LIN {X 0,Y 366.186,Z 582.317,A -85,B 0,C 180,E1 11317.948,E2 11317.948} C_VEL
LIN {X 0,Y 371.431,Z 589.202,A -85,B 0,C 180,E1 11315.424,E2 11315.424} C_VEL
LIN {X 0,Y 378.008,Z 597.97,A -85,B 0,C 180,E1 11312.682,E2 11312.682} C_VEL
LIN {X 0,Y 385.262,Z 608.266,A -85,B 0,C 180,E1 11310.027,E2 11310.027} C_VEL
LIN {X 0,Y 392.759,Z 619.158,A -85,B 0,C 180,E1 11307.596,E2 11307.596} C_VEL
LIN {X 0,Y 401.924,Z 633.691,A -85,B 0,C 180,E1 11304.924,E2 11304.924} C_VEL
LIN {X 0,Y 408.714,Z 645.3,A -85,B 0,C 180,E1 11303.115,E2 11303.115} C_VEL
LIN {X 0,Y 397.678,Z 876.786,A -85,B 0,C 180,E1 11298.792,E2 11298.792} C_VEL
LIN {X 0,Y 395.952,Z 903.504,A -85,B 0,C 180,E1 11298.228,E2 11298.228} C_VEL
LIN {X 0,Y 393.493,Z 925.311,A -85,B 0,C 180,E1 11297.568,E2 11297.568} C_VEL
LIN {X 0,Y 390.28,Z 946.189,A -85,B 0,C 180,E1 11296.684,E2 11296.684} C_VEL
LIN {X 0,Y 386.282,Z 967.256,A -85,B 0,C 180,E1 11295.529,E2 11295.529} C_VEL
LIN {X 0,Y 382.072,Z 986.142,A -85,B 0,C 180,E1 11294.243,E2 11294.243} C_VEL
LIN {X 0,Y 377.137,Z 1005.209,A -85,B 0,C 180,E1 11292.639,E2 11292.639} C_VEL
LIN {X 0,Y 371.736,Z 1024.131,A -85,B 0,C 180,E1 11290.712,E2 11290.712} C_VEL
LIN {X 0,Y 366.371,Z 1041.49,A -85,B 0,C 180,E1 11288.579,E2 11288.579} C_VEL
LIN {X 0,Y 361.104,Z 1057.311,A -85,B 0,C 180,E1 11286.24,E2 11286.24} C_VEL
LIN {X 0,Y 355.944,Z 1072.38,A -85,B 0,C 180,E1 11283.599,E2 11283.599} C_VEL
LIN {X 0,Y 351.082,Z 1086.425,A -85,B 0,C 180,E1 11280.649,E2 11280.649} C_VEL
LIN {X 0,Y 346.966,Z 1098.332,A -85,B 0,C 180,E1 11277.643,E2 11277.643} C_VEL
LIN {X 0,Y 343.299,Z 1109.594,A -85,B 0,C 180,E1 11274.247,E2 11274.247} C_VEL
LIN {X 0,Y 340.505,Z 1118.917,A -85,B 0,C 180,E1 11270.812,E2 11270.812} C_VEL
LIN {X 0,Y 338.432,Z 1126.851,A -85,B 0,C 180,E1 11267.184,E2 11267.184} C_VEL
LIN {X 0,Y 337.113,Z 1133.168,A -85,B 0,C 180,E1 11263.551,E2 11263.551} C_VEL
LIN {X 0,Y 336.408,Z 1137.619,A -85,B 0,C 180,E1 11260.099,E2 11260.099} C_VEL
LIN {X 0,Y 336.159,Z 1139.83,A -85,B 0,C 180,E1 11257.841,E2 11257.841} C_VEL
LIN {X 0,Y 335.071,Z 1140.944,A -85,B 0,C 180,E1 11256.542,E2 11256.542} C_VEL
LIN {X 0,Y 330.367,Z 1142.612,A -85,B 0,C 180,E1 11254.081,E2 11254.081} C_VEL
LIN {X 0,Y 328.115,Z 1143.242,A -85,B 0,C 180,E1 11252.372,E2 11252.372} C_VEL
LIN {X 0,Y 327.966,Z 1143.315,A -85,B 0,C 180,E1 11251.884,E2 11251.884} C_VEL
LIN {X 0,Y 327.969,Z 1143.385,A -85,B 0,C 180,E1 11248.602,E2 11248.602} C_VEL
LIN {X 0,Y 328.018,Z 1142.229,A -85,B 0,C 180,E1 11244.929,E2 11244.929} C_VEL
LIN {X 0,Y 328.248,Z 1139.737,A -85,B 0,C 180,E1 11241.416,E2 11241.416} C_VEL
LIN {X 0,Y 328.872,Z 1135.354,A -85,B 0,C 180,E1 11237.404,E2 11237.404} C_VEL
LIN {X 0,Y 330.06,Z 1129.659,A -85,B 0,C 180,E1 11233.637,E2 11233.637} C_VEL
LIN {X 0,Y 331.98,Z 1122.268,A -85,B 0,C 180,E1 11229.919,E2 11229.919} C_VEL
LIN {X 0,Y 334.944,Z 1112.65,A -85,B 0,C 180,E1 11226.047,E2 11226.047} C_VEL
LIN {X 0,Y 338.59,Z 1102.053,A -85,B 0,C 180,E1 11222.57,E2 11222.57} C_VEL
LIN {X 0,Y 342.919,Z 1089.92,A -85,B 0,C 180,E1 11219.319,E2 11219.319} C_VEL
LIN {X 0,Y 347.843,Z 1076.454,A -85,B 0,C 180,E1 11216.305,E2 11216.305} C_VEL
LIN {X 0,Y 353.24,Z 1061.666,A -85,B 0,C 180,E1 11213.529,E2 11213.529} C_VEL
LIN {X 0,Y 358.581,Z 1046.318,A -85,B 0,C 180,E1 11211.142,E2 11211.142} C_VEL
LIN {X 0,Y 364.459,Z 1028.526,A -85,B 0,C 180,E1 11208.82,E2 11208.82} C_VEL
LIN {X 0,Y 370.03,Z 1010.354,A -85,B 0,C 180,E1 11206.851,E2 11206.851} C_VEL
LIN {X 0,Y 375.194,Z 991.424,A -85,B 0,C 180,E1 11205.181,E2 11205.181} C_VEL
LIN {X 0,Y 380.213,Z 970.596,A -85,B 0,C 180,E1 11203.682,E2 11203.682} C_VEL
LIN {X 0,Y 384.198,Z 951.289,A -85,B 0,C 180,E1 11202.566,E2 11202.566} C_VEL
LIN {X 0,Y 387.659,Z 930.348,A -85,B 0,C 180,E1 11201.626,E2 11201.626} C_VEL
LIN {X 0,Y 390.429,Z 909.023,A -85,B 0,C 180,E1 11200.912,E2 11200.912} C_VEL
LIN {X 0,Y 392.234,Z 887.054,A -85,B 0,C 180,E1 11200.398,E2 11200.398} C_VEL
LIN {X 0,Y 400.836,Z 709.616,A -85,B 0,C 180,E1 11197.043,E2 11197.043} C_VEL
LIN {X 0,Y 396.954,Z 714.225,A -85,B 0,C 180,E1 11196.361,E2 11196.361} C_VEL
LIN {X 0,Y 391.32,Z 723.362,A -85,B 0,C 180,E1 11195.402,E2 11195.402} C_VEL
LIN {X 0,Y 386.047,Z 730.128,A -85,B 0,C 180,E1 11194.399,E2 11194.399} C_VEL
LIN {X 0,Y 380.733,Z 739.752,A -85,B 0,C 180,E1 11193.425,E2 11193.425} C_VEL
LIN {X 0,Y 377.937,Z 744.145,A -85,B 0,C 180,E1 11192.866,E2 11192.866} C_VEL
LIN {X 0,Y 373.251,Z 764.172,A -85,B 0,C 180,E1 11192.35,E2 11192.35} C_VEL
LIN {X 0,Y 369.775,Z 775.752,A -85,B 0,C 180,E1 11191.833,E2 11191.833} C_VEL
LIN {X 0,Y 367.625,Z 781.787,A -85,B 0,C 180,E1 11191.463,E2 11191.463} C_VEL
LIN {X 0,Y 361.181,Z 811.219,A -85,B 0,C 180,E1 11190.749,E2 11190.749} C_VEL
LIN {X 0,Y 357.761,Z 823.668,A -85,B 0,C 180,E1 11190.226,E2 11190.226} C_VEL
LIN {X 0,Y 354.98,Z 831.573,A -85,B 0,C 180,E1 11189.695,E2 11189.695} C_VEL
LIN {X 0,Y 348.335,Z 862.323,A -85,B 0,C 180,E1 11188.874,E2 11188.874} C_VEL
LIN {X 0,Y 345.171,Z 873.899,A -85,B 0,C 180,E1 11188.328,E2 11188.328} C_VEL
LIN {X 0,Y 343.261,Z 880.377,A -85,B 0,C 180,E1 11187.812,E2 11187.812} C_VEL
LIN {X 0,Y 342.63,Z 889.884,A -85,B 0,C 180,E1 11187.433,E2 11187.433} C_VEL
LIN {X 0,Y 342.059,Z 911.963,A -85,B 0,C 180,E1 11186.73,E2 11186.73} C_VEL
LIN {X 0,Y 341.208,Z 929.996,A -85,B 0,C 180,E1 11185.842,E2 11185.842} C_VEL
LIN {X 0,Y 339.993,Z 948.311,A -85,B 0,C 180,E1 11184.591,E2 11184.591} C_VEL
LIN {X 0,Y 338.687,Z 963.946,A -85,B 0,C 180,E1 11183.211,E2 11183.211} C_VEL
LIN {X 0,Y 337.194,Z 979.445,A -85,B 0,C 180,E1 11181.482,E2 11181.482} C_VEL
LIN {X 0,Y 335.66,Z 993.949,A -85,B 0,C 180,E1 11179.489,E2 11179.489} C_VEL
LIN {X 0,Y 334.281,Z 1006.231,A -85,B 0,C 180,E1 11177.404,E2 11177.404} C_VEL
LIN {X 0,Y 332.98,Z 1017.915,A -85,B 0,C 180,E1 11174.966,E2 11174.966} C_VEL
LIN {X 0,Y 332,Z 1027.395,A -85,B 0,C 180,E1 11172.524,E2 11172.524} C_VEL
LIN {X 0,Y 331.241,Z 1035.395,A -85,B 0,C 180,E1 11169.908,E2 11169.908} C_VEL
LIN {X 0,Y 330.761,Z 1041.946,A -85,B 0,C 180,E1 11167.12,E2 11167.12} C_VEL
LIN {X 0,Y 330.565,Z 1046.667,A -85,B 0,C 180,E1 11164.337,E2 11164.337} C_VEL
LIN {X 0,Y 330.581,Z 1049.61,A -85,B 0,C 180,E1 11161.56,E2 11161.56} C_VEL
LIN {X 0,Y 330.804,Z 1050.944,A -85,B 0,C 180,E1 11158.615,E2 11158.615} C_VEL
LIN {X 0,Y 331.202,Z 1050.526,A -85,B 0,C 180,E1 11155.846,E2 11155.846} C_VEL
LIN {X 0,Y 331.838,Z 1048.398,A -85,B 0,C 180,E1 11153.078,E2 11153.078} C_VEL
LIN {X 0,Y 332.756,Z 1044.468,A -85,B 0,C 180,E1 11150.313,E2 11150.313} C_VEL
LIN {X 0,Y 334.013,Z 1038.61,A -85,B 0,C 180,E1 11147.554,E2 11147.554} C_VEL
LIN {X 0,Y 335.392,Z 1031.672,A -85,B 0,C 180,E1 11145.145,E2 11145.145} C_VEL
LIN {X 0,Y 337.024,Z 1022.654,A -85,B 0,C 180,E1 11142.743,E2 11142.743} C_VEL
LIN {X 0,Y 338.799,Z 1012.138,A -85,B 0,C 180,E1 11140.52,E2 11140.52} C_VEL
LIN {X 0,Y 340.605,Z 999.902,A -85,B 0,C 180,E1 11138.473,E2 11138.473} C_VEL
LIN {X 0,Y 342.308,Z 986.562,A -85,B 0,C 180,E1 11136.686,E2 11136.686} C_VEL
LIN {X 0,Y 343.887,Z 971.383,A -85,B 0,C 180,E1 11135.066,E2 11135.066} C_VEL
LIN {X 0,Y 345.235,Z 954.859,A -85,B 0,C 180,E1 11133.698,E2 11133.698} C_VEL
LIN {X 0,Y 346.219,Z 937.734,A -85,B 0,C 180,E1 11132.62,E2 11132.62} C_VEL
LIN {X 0,Y 346.855,Z 927.468,A -85,B 0,C 180,E1 11132.068,E2 11132.068} C_VEL
LIN {X 0,Y 348,Z 924.934,A -85,B 0,C 180,E1 11131.772,E2 11131.772} C_VEL
LIN {X 0,Y 350.86,Z 920.539,A -85,B 0,C 180,E1 11131.345,E2 11131.345} C_VEL
LIN {X 0,Y 354.501,Z 912.006,A -85,B 0,C 180,E1 11131.007,E2 11131.007} C_VEL
LIN {X 0,Y 357.108,Z 904.907,A -85,B 0,C 180,E1 11130.799,E2 11130.799} C_VEL
LIN {X 0,Y 360.337,Z 898.788,A -85,B 0,C 180,E1 11130.331,E2 11130.331} C_VEL
LIN {X 0,Y 363.987,Z 888.542,A -85,B 0,C 180,E1 11129.925,E2 11129.925} C_VEL
LIN {X 0,Y 369.949,Z 866.042,A -85,B 0,C 180,E1 11129.35,E2 11129.35} C_VEL
LIN {X 0,Y 373.838,Z 855.883,A -85,B 0,C 180,E1 11128.8,E2 11128.8} C_VEL
LIN {X 0,Y 378.866,Z 838.681,A -85,B 0,C 180,E1 11128.259,E2 11128.259} C_VEL
LIN {X 0,Y 383.059,Z 822.695,A -85,B 0,C 180,E1 11127.883,E2 11127.883} C_VEL
LIN {X 0,Y 387.383,Z 811.4,A -85,B 0,C 180,E1 11127.333,E2 11127.333} C_VEL
LIN {X 0,Y 392.621,Z 793.713,A -85,B 0,C 180,E1 11126.825,E2 11126.825} C_VEL
LIN {X 0,Y 396.512,Z 779.247,A -85,B 0,C 180,E1 11126.502,E2 11126.502} C_VEL
LIN {X 0,Y 399.615,Z 771.69,A -85,B 0,C 180,E1 11126.126,E2 11126.126} C_VEL
LIN {X 0,Y 392.671,Z 892.302,A -85,B 0,C 180,E1 11123.671,E2 11123.671} C_VEL
LIN {X 0,Y 390.102,Z 915.62,A -85,B 0,C 180,E1 11123.008,E2 11123.008} C_VEL
LIN {X 0,Y 386.994,Z 937.185,A -85,B 0,C 180,E1 11122.181,E2 11122.181} C_VEL
LIN {X 0,Y 382.98,Z 959.044,A -85,B 0,C 180,E1 11121.078,E2 11121.078} C_VEL
LIN {X 0,Y 378.27,Z 980.989,A -85,B 0,C 180,E1 11119.696,E2 11119.696} C_VEL
LIN {X 0,Y 373.314,Z 1001.28,A -85,B 0,C 180,E1 11118.123,E2 11118.123} C_VEL
LIN {X 0,Y 367.979,Z 1020.909,A -85,B 0,C 180,E1 11116.284,E2 11116.284} C_VEL
LIN {X 0,Y 362.493,Z 1039.821,A -85,B 0,C 180,E1 11114.181,E2 11114.181} C_VEL
LIN {X 0,Y 356.917,Z 1057.605,A -85,B 0,C 180,E1 11111.815,E2 11111.815} C_VEL
LIN {X 0,Y 351.301,Z 1075.094,A -85,B 0,C 180,E1 11109.082,E2 11109.082} C_VEL
LIN {X 0,Y 346.378,Z 1090.22,A -85,B 0,C 180,E1 11106.282,E2 11106.282} C_VEL
LIN {X 0,Y 341.513,Z 1105.32,A -85,B 0,C 180,E1 11102.995,E2 11102.995} C_VEL
LIN {X 0,Y 337.534,Z 1118.368,A -85,B 0,C 180,E1 11099.65,E2 11099.65} C_VEL
LIN {X 0,Y 334.214,Z 1129.964,A -85,B 0,C 180,E1 11096.09,E2 11096.09} C_VEL
LIN {X 0,Y 331.63,Z 1140.317,A -85,B 0,C 180,E1 11092.327,E2 11092.327} C_VEL
LIN {X 0,Y 329.914,Z 1148.379,A -85,B 0,C 180,E1 11088.739,E2 11088.739} C_VEL
LIN {X 0,Y 328.748,Z 1155.565,A -85,B 0,C 180,E1 11084.802,E2 11084.802} C_VEL
LIN {X 0,Y 328.211,Z 1160.559,A -85,B 0,C 180,E1 11081.209,E2 11081.209} C_VEL
LIN {X 0,Y 327.959,Z 1164.449,A -85,B 0,C 180,E1 11077.357,E2 11077.357} C_VEL
LIN {X 0,Y 327.941,Z 1166.518,A -85,B 0,C 180,E1 11073.846,E2 11073.846} C_VEL
LIN {X 0,Y 327.936,Z 1167.332,A -85,B 0,C 180,E1 11070.524,E2 11070.524} C_VEL
LIN {X 0,Y 327.927,Z 1166.805,A -85,B 0,C 180,E1 11066.854,E2 11066.854} C_VEL
LIN {X 0,Y 327.965,Z 1165.053,A -85,B 0,C 180,E1 11063.523,E2 11063.523} C_VEL
LIN {X 0,Y 328.1,Z 1161.814,A -85,B 0,C 180,E1 11059.819,E2 11059.819} C_VEL
LIN {X 0,Y 328.575,Z 1156.905,A -85,B 0,C 180,E1 11056.09,E2 11056.09} C_VEL
LIN {X 0,Y 329.54,Z 1150.522,A -85,B 0,C 180,E1 11052.307,E2 11052.307} C_VEL
LIN {X 0,Y 331.12,Z 1142.434,A -85,B 0,C 180,E1 11048.569,E2 11048.569} C_VEL
LIN {X 0,Y 333.509,Z 1132.644,A -85,B 0,C 180,E1 11044.804,E2 11044.804} C_VEL
LIN {X 0,Y 336.436,Z 1121.99,A -85,B 0,C 180,E1 11041.414,E2 11041.414} C_VEL
LIN {X 0,Y 340.395,Z 1108.935,A -85,B 0,C 180,E1 11037.882,E2 11037.882} C_VEL
LIN {X 0,Y 344.735,Z 1095.225,A -85,B 0,C 180,E1 11034.748,E2 11034.748} C_VEL
LIN {X 0,Y 349.892,Z 1079.355,A -85,B 0,C 180,E1 11031.676,E2 11031.676} C_VEL
LIN {X 0,Y 355.227,Z 1062.965,A -85,B 0,C 180,E1 11028.967,E2 11028.967} C_VEL
LIN {X 0,Y 360.826,Z 1044.991,A -85,B 0,C 180,E1 11026.48,E2 11026.48} C_VEL
LIN {X 0,Y 366.707,Z 1025.329,A -85,B 0,C 180,E1 11024.185,E2 11024.185} C_VEL
LIN {X 0,Y 371.762,Z 1007.076,A -85,B 0,C 180,E1 11022.396,E2 11022.396} C_VEL
LIN {X 0,Y 377.049,Z 986.011,A -85,B 0,C 180,E1 11020.675,E2 11020.675} C_VEL
LIN {X 0,Y 381.795,Z 964.869,A -85,B 0,C 180,E1 11019.258,E2 11019.258} C_VEL
LIN {X 0,Y 385.904,Z 942.947,A -85,B 0,C 180,E1 11018.093,E2 11018.093} C_VEL
LIN {X 0,Y 389.526,Z 919.577,A -85,B 0,C 180,E1 11017.128,E2 11017.128} C_VEL
LIN {X 0,Y 392.156,Z 897.248,A -85,B 0,C 180,E1 11016.458,E2 11016.458} C_VEL
LIN {X 0,Y 394.386,Z 863.932,A -85,B 0,C 180,E1 11015.736,E2 11015.736} C_VEL
LIN {X 0,Y 406.266,Z 655.335,A -85,B 0,C 180,E1 11011.555,E2 11011.555} C_VEL
LIN {X 0,Y 406.902,Z 643.594,A -85,B 0,C 180,E1 11011.312,E2 11011.312} C_VEL
LIN {X 0,Y 397.581,Z 629.012,A -85,B 0,C 180,E1 11008.748,E2 11008.748} C_VEL
LIN {X 0,Y 388.35,Z 615.637,A -85,B 0,C 180,E1 11005.915,E2 11005.915} C_VEL
LIN {X 0,Y 380.432,Z 605.01,A -85,B 0,C 180,E1 11003.177,E2 11003.177} C_VEL
LIN {X 0,Y 373.333,Z 595.852,A -85,B 0,C 180,E1 11000.375,E2 11000.375} C_VEL
LIN {X 0,Y 368.267,Z 589.841,A -85,B 0,C 180,E1 10998.111,E2 10998.111} C_VEL
LIN {X 0,Y 363.853,Z 584.59,A -85,B 0,C 180,E1 10995.868,E2 10995.868} C_VEL
LIN {X 0,Y 358.835,Z 578.864,A -85,B 0,C 180,E1 10992.88,E2 10992.88} C_VEL
LIN {X 0,Y 353.311,Z 572.841,A -85,B 0,C 180,E1 10988.626,E2 10988.626} C_VEL
LIN {X 0,Y 348.081,Z 567.999,A -85,B 0,C 180,E1 10981.646,E2 10981.646} C_VEL
LIN {X 0,Y 347.245,Z 567.182,A -85,B 0,C 180,E1 10978.184,E2 10978.184} C_VEL
LIN {X 0,Y 347.496,Z 568.254,A -85,B 0,C 180,E1 10974.551,E2 10974.551} C_VEL
LIN {X 0,Y 351.064,Z 572.556,A -85,B 0,C 180,E1 10968.166,E2 10968.166} C_VEL
LIN {X 0,Y 354.487,Z 577.164,A -85,B 0,C 180,E1 10964.792,E2 10964.792} C_VEL
LIN {X 0,Y 355.794,Z 578.575,A -85,B 0,C 180,E1 10963.762,E2 10963.762} C_VEL
LIN {X 0,Y 359.364,Z 583.21,A -85,B 0,C 180,E1 10961.255,E2 10961.255} C_VEL
LIN {X 0,Y 364.436,Z 589.819,A -85,B 0,C 180,E1 10958.303,E2 10958.303} C_VEL
LIN {X 0,Y 369.585,Z 596.701,A -85,B 0,C 180,E1 10955.761,E2 10955.761} C_VEL
LIN {X 0,Y 376.05,Z 605.555,A -85,B 0,C 180,E1 10952.999,E2 10952.999} C_VEL
LIN {X 0,Y 382.814,Z 615.312,A -85,B 0,C 180,E1 10950.462,E2 10950.462} C_VEL
LIN {X 0,Y 389.968,Z 625.925,A -85,B 0,C 180,E1 10948.076,E2 10948.076} C_VEL
LIN {X 0,Y 398.766,Z 640.106,A -85,B 0,C 180,E1 10945.438,E2 10945.438} C_VEL
LIN {X 0,Y 404.034,Z 649.281,A -85,B 0,C 180,E1 10943.979,E2 10943.979} C_VEL
LIN {X 0,Y 392.554,Z 879.807,A -85,B 0,C 180,E1 10939.647,E2 10939.647} C_VEL
LIN {X 0,Y 390.832,Z 904.21,A -85,B 0,C 180,E1 10939.118,E2 10939.118} C_VEL
LIN {X 0,Y 388.219,Z 926.195,A -85,B 0,C 180,E1 10938.44,E2 10938.44} C_VEL
LIN {X 0,Y 384.946,Z 946.674,A -85,B 0,C 180,E1 10937.567,E2 10937.567} C_VEL
LIN {X 0,Y 380.888,Z 967.279,A -85,B 0,C 180,E1 10936.429,E2 10936.429} C_VEL
LIN {X 0,Y 376.38,Z 986.786,A -85,B 0,C 180,E1 10935.094,E2 10935.094} C_VEL
LIN {X 0,Y 371.267,Z 1005.752,A -85,B 0,C 180,E1 10933.479,E2 10933.479} C_VEL
LIN {X 0,Y 365.653,Z 1024.604,A -85,B 0,C 180,E1 10931.537,E2 10931.537} C_VEL
LIN {X 0,Y 360.07,Z 1041.94,A -85,B 0,C 180,E1 10929.384,E2 10929.384} C_VEL
LIN {X 0,Y 354.594,Z 1057.668,A -85,B 0,C 180,E1 10927.024,E2 10927.024} C_VEL
LIN {X 0,Y 349.176,Z 1072.757,A -85,B 0,C 180,E1 10924.34,E2 10924.34} C_VEL
LIN {X 0,Y 344.328,Z 1086.047,A -85,B 0,C 180,E1 10921.513,E2 10921.513} C_VEL
LIN {X 0,Y 339.729,Z 1098.679,A -85,B 0,C 180,E1 10918.284,E2 10918.284} C_VEL
LIN {X 0,Y 335.848,Z 1109.925,A -85,B 0,C 180,E1 10914.82,E2 10914.82} C_VEL
LIN {X 0,Y 332.874,Z 1119.245,A -85,B 0,C 180,E1 10911.312,E2 10911.312} C_VEL
LIN {X 0,Y 330.651,Z 1127.166,A -85,B 0,C 180,E1 10907.601,E2 10907.601} C_VEL
LIN {X 0,Y 329.229,Z 1133.474,A -85,B 0,C 180,E1 10903.882,E2 10903.882} C_VEL
LIN {X 0,Y 328.457,Z 1137.92,A -85,B 0,C 180,E1 10900.347,E2 10900.347} C_VEL
LIN {X 0,Y 328.095,Z 1141.313,A -85,B 0,C 180,E1 10896.474,E2 10896.474} C_VEL
LIN {X 0,Y 327.975,Z 1143.026,A -85,B 0,C 180,E1 10892.971,E2 10892.971} C_VEL
LIN {X 0,Y 327.966,Z 1143.315,A -85,B 0,C 180,E1 10891.884,E2 10891.884} C_VEL
LIN {X 0,Y 326.958,Z 1143.526,A -85,B 0,C 180,E1 10890.538,E2 10890.538} C_VEL
LIN {X 0,Y 322.684,Z 1143.537,A -85,B 0,C 180,E1 10888.184,E2 10888.184} C_VEL
LIN {X 0,Y 320.264,Z 1143.171,A -85,B 0,C 180,E1 10886.435,E2 10886.435} C_VEL
LIN {X 0,Y 320.013,Z 1142.918,A -85,B 0,C 180,E1 10885.736,E2 10885.736} C_VEL
LIN {X 0,Y 320.204,Z 1140.562,A -85,B 0,C 180,E1 10881.834,E2 10881.834} C_VEL
LIN {X 0,Y 320.744,Z 1136.958,A -85,B 0,C 180,E1 10878.127,E2 10878.127} C_VEL
LIN {X 0,Y 321.813,Z 1131.693,A -85,B 0,C 180,E1 10874.317,E2 10874.317} C_VEL
LIN {X 0,Y 323.691,Z 1124.701,A -85,B 0,C 180,E1 10870.412,E2 10870.412} C_VEL
LIN {X 0,Y 326.349,Z 1116.278,A -85,B 0,C 180,E1 10866.72,E2 10866.72} C_VEL
LIN {X 0,Y 329.869,Z 1106.265,A -85,B 0,C 180,E1 10863.151,E2 10863.151} C_VEL
LIN {X 0,Y 334.125,Z 1095.008,A -85,B 0,C 180,E1 10859.819,E2 10859.819} C_VEL
LIN {X 0,Y 338.965,Z 1082.307,A -85,B 0,C 180,E1 10856.725,E2 10856.725} C_VEL
LIN {X 0,Y 344.643,Z 1067.47,A -85,B 0,C 180,E1 10853.713,E2 10853.713} C_VEL
LIN {X 0,Y 350.375,Z 1052.151,A -85,B 0,C 180,E1 10851.111,E2 10851.111} C_VEL
LIN {X 0,Y 356.201,Z 1035.575,A -85,B 0,C 180,E1 10848.789,E2 10848.789} C_VEL
LIN {X 0,Y 362.114,Z 1017.486,A -85,B 0,C 180,E1 10846.674,E2 10846.674} C_VEL
LIN {X 0,Y 367.65,Z 999.07,A -85,B 0,C 180,E1 10844.89,E2 10844.89} C_VEL
LIN {X 0,Y 372.724,Z 979.661,A -85,B 0,C 180,E1 10843.366,E2 10843.366} C_VEL
LIN {X 0,Y 377.633,Z 958.028,A -85,B 0,C 180,E1 10842.001,E2 10842.001} C_VEL
LIN {X 0,Y 381.486,Z 937.643,A -85,B 0,C 180,E1 10840.989,E2 10840.989} C_VEL
LIN {X 0,Y 384.509,Z 916.783,A -85,B 0,C 180,E1 10840.216,E2 10840.216} C_VEL
LIN {X 0,Y 386.877,Z 893.893,A -85,B 0,C 180,E1 10839.609,E2 10839.609} C_VEL
LIN {X 0,Y 395.423,Z 726.724,A -85,B 0,C 180,E1 10836.412,E2 10836.412} C_VEL
LIN {X 0,Y 389.741,Z 734.274,A -85,B 0,C 180,E1 10835.391,E2 10835.391} C_VEL
LIN {X 0,Y 388.254,Z 736.358,A -85,B 0,C 180,E1 10835.118,E2 10835.118} C_VEL
LIN {X 0,Y 382.655,Z 746.09,A -85,B 0,C 180,E1 10834.112,E2 10834.112} C_VEL
LIN {X 0,Y 381.204,Z 748.533,A -85,B 0,C 180,E1 10833.84,E2 10833.84} C_VEL
LIN {X 0,Y 376.48,Z 768.015,A -85,B 0,C 180,E1 10833.328,E2 10833.328} C_VEL
LIN {X 0,Y 372.844,Z 779.678,A -85,B 0,C 180,E1 10832.8,E2 10832.8} C_VEL
LIN {X 0,Y 370.943,Z 785.021,A -85,B 0,C 180,E1 10832.489,E2 10832.489} C_VEL
LIN {X 0,Y 364.868,Z 812.647,A -85,B 0,C 180,E1 10831.855,E2 10831.855} C_VEL
LIN {X 0,Y 361.186,Z 826.037,A -85,B 0,C 180,E1 10831.327,E2 10831.327} C_VEL
LIN {X 0,Y 358.041,Z 835.013,A -85,B 0,C 180,E1 10830.763,E2 10830.763} C_VEL
LIN {X 0,Y 351.854,Z 863.566,A -85,B 0,C 180,E1 10830.045,E2 10830.045} C_VEL
LIN {X 0,Y 348.377,Z 876.333,A -85,B 0,C 180,E1 10829.487,E2 10829.487} C_VEL
LIN {X 0,Y 345.584,Z 884.318,A -85,B 0,C 180,E1 10828.929,E2 10828.929} C_VEL
LIN {X 0,Y 340.968,Z 902.377,A -85,B 0,C 180,E1 10828.421,E2 10828.421} C_VEL
LIN {X 0,Y 338.111,Z 910.025,A -85,B 0,C 180,E1 10827.999,E2 10827.999} C_VEL
LIN {X 0,Y 335.704,Z 914.211,A -85,B 0,C 180,E1 10827.494,E2 10827.494} C_VEL
LIN {X 0,Y 334.698,Z 916.443,A -85,B 0,C 180,E1 10827.145,E2 10827.145} C_VEL
LIN {X 0,Y 334.105,Z 923.12,A -85,B 0,C 180,E1 10826.71,E2 10826.71} C_VEL
LIN {X 0,Y 333.011,Z 940.969,A -85,B 0,C 180,E1 10825.618,E2 10825.618} C_VEL
LIN {X 0,Y 331.715,Z 957.602,A -85,B 0,C 180,E1 10824.292,E2 10824.292} C_VEL
LIN {X 0,Y 330.271,Z 973.167,A -85,B 0,C 180,E1 10822.706,E2 10822.706} C_VEL
LIN {X 0,Y 328.644,Z 988.624,A -85,B 0,C 180,E1 10820.747,E2 10820.747} C_VEL
LIN {X 0,Y 327.133,Z 1002.002,A -85,B 0,C 180,E1 10818.649,E2 10818.649} C_VEL
LIN {X 0,Y 325.686,Z 1014.514,A -85,B 0,C 180,E1 10816.223,E2 10816.223} C_VEL
LIN {X 0,Y 324.541,Z 1024.958,A -85,B 0,C 180,E1 10813.723,E2 10813.723} C_VEL
LIN {X 0,Y 323.627,Z 1033.816,A -85,B 0,C 180,E1 10811.044,E2 10811.044} C_VEL
LIN {X 0,Y 323.014,Z 1041.171,A -85,B 0,C 180,E1 10808.187,E2 10808.187} C_VEL
LIN {X 0,Y 322.715,Z 1046.589,A -85,B 0,C 180,E1 10805.334,E2 10805.334} C_VEL
LIN {X 0,Y 322.669,Z 1050.192,A -85,B 0,C 180,E1 10802.487,E2 10802.487} C_VEL
LIN {X 0,Y 322.84,Z 1052.161,A -85,B 0,C 180,E1 10799.646,E2 10799.646} C_VEL
LIN {X 0,Y 323.2,Z 1052.49,A -85,B 0,C 180,E1 10796.808,E2 10796.808} C_VEL
LIN {X 0,Y 323.787,Z 1051.094,A -85,B 0,C 180,E1 10793.974,E2 10793.974} C_VEL
LIN {X 0,Y 324.668,Z 1047.947,A -85,B 0,C 180,E1 10791.143,E2 10791.143} C_VEL
LIN {X 0,Y 325.807,Z 1043.336,A -85,B 0,C 180,E1 10788.494,E2 10788.494} C_VEL
LIN {X 0,Y 327.257,Z 1036.876,A -85,B 0,C 180,E1 10785.853,E2 10785.853} C_VEL
LIN {X 0,Y 328.888,Z 1028.915,A -85,B 0,C 180,E1 10783.396,E2 10783.396} C_VEL
LIN {X 0,Y 330.818,Z 1018.72,A -85,B 0,C 180,E1 10780.949,E2 10780.949} C_VEL
LIN {X 0,Y 332.691,Z 1007.755,A -85,B 0,C 180,E1 10778.861,E2 10778.861} C_VEL
LIN {X 0,Y 334.725,Z 993.982,A -85,B 0,C 180,E1 10776.778,E2 10776.778} C_VEL
LIN {X 0,Y 336.414,Z 980.305,A -85,B 0,C 180,E1 10775.131,E2 10775.131} C_VEL
LIN {X 0,Y 338.044,Z 963.928,A -85,B 0,C 180,E1 10773.568,E2 10773.568} C_VEL
LIN {X 0,Y 339.554,Z 945.986,A -85,B 0,C 180,E1 10772.226,E2 10772.226} C_VEL
LIN {X 0,Y 341.095,Z 943.634,A -85,B 0,C 180,E1 10771.84,E2 10771.84} C_VEL
LIN {X 0,Y 343.848,Z 940.297,A -85,B 0,C 180,E1 10771.423,E2 10771.423} C_VEL
LIN {X 0,Y 347.469,Z 933.968,A -85,B 0,C 180,E1 10771.059,E2 10771.059} C_VEL
LIN {X 0,Y 349.146,Z 930.779,A -85,B 0,C 180,E1 10770.894,E2 10770.894} C_VEL
LIN {X 0,Y 352.778,Z 925.763,A -85,B 0,C 180,E1 10770.382,E2 10770.382} C_VEL
LIN {X 0,Y 356.445,Z 918.319,A -85,B 0,C 180,E1 10770.026,E2 10770.026} C_VEL
LIN {X 0,Y 360.184,Z 908.815,A -85,B 0,C 180,E1 10769.769,E2 10769.769} C_VEL
LIN {X 0,Y 363.94,Z 901.445,A -85,B 0,C 180,E1 10769.27,E2 10769.27} C_VEL
LIN {X 0,Y 367.943,Z 890.444,A -85,B 0,C 180,E1 10768.875,E2 10768.875} C_VEL
LIN {X 0,Y 373.651,Z 869.308,A -85,B 0,C 180,E1 10768.367,E2 10768.367} C_VEL
LIN {X 0,Y 377.881,Z 858.203,A -85,B 0,C 180,E1 10767.804,E2 10767.804} C_VEL
LIN {X 0,Y 383.109,Z 840.443,A -85,B 0,C 180,E1 10767.273,E2 10767.273} C_VEL
LIN {X 0,Y 386.977,Z 825.805,A -85,B 0,C 180,E1 10766.942,E2 10766.942} C_VEL
LIN {X 0,Y 391.552,Z 813.854,A -85,B 0,C 180,E1 10766.393,E2 10766.393} C_VEL
LIN {X 0,Y 392.634,Z 810.634,A -85,B 0,C 180,E1 10766.279,E2 10766.279} C_VEL
LIN {X 0,Y 387.642,Z 893.325,A -85,B 0,C 180,E1 10764.575,E2 10764.575} C_VEL
LIN {X 0,Y 384.969,Z 916.404,A -85,B 0,C 180,E1 10763.908,E2 10763.908} C_VEL
LIN {X 0,Y 381.619,Z 938.498,A -85,B 0,C 180,E1 10763.046,E2 10763.046} C_VEL
LIN {X 0,Y 377.693,Z 959.165,A -85,B 0,C 180,E1 10761.994,E2 10761.994} C_VEL
LIN {X 0,Y 372.733,Z 981.395,A -85,B 0,C 180,E1 10760.585,E2 10760.585} C_VEL
LIN {X 0,Y 367.606,Z 1001.596,A -85,B 0,C 180,E1 10759.006,E2 10759.006} C_VEL
LIN {X 0,Y 361.839,Z 1021.894,A -85,B 0,C 180,E1 10757.077,E2 10757.077} C_VEL
LIN {X 0,Y 356.217,Z 1040.431,A -85,B 0,C 180,E1 10754.982,E2 10754.982} C_VEL
LIN {X 0,Y 350.348,Z 1058.306,A -85,B 0,C 180,E1 10752.561,E2 10752.561} C_VEL
LIN {X 0,Y 344.265,Z 1076.277,A -85,B 0,C 180,E1 10749.679,E2 10749.679} C_VEL
LIN {X 0,Y 339.058,Z 1091.573,A -85,B 0,C 180,E1 10746.772,E2 10746.772} C_VEL
LIN {X 0,Y 334.241,Z 1105.676,A -85,B 0,C 180,E1 10743.602,E2 10743.602} C_VEL
LIN {X 0,Y 330.064,Z 1118.655,A -85,B 0,C 180,E1 10740.19,E2 10740.19} C_VEL
LIN {X 0,Y 326.561,Z 1130.155,A -85,B 0,C 180,E1 10736.553,E2 10736.553} C_VEL
LIN {X 0,Y 323.722,Z 1140.835,A -85,B 0,C 180,E1 10732.519,E2 10732.519} C_VEL
LIN {X 0,Y 322.021,Z 1148.425,A -85,B 0,C 180,E1 10729.027,E2 10729.027} C_VEL
LIN {X 0,Y 320.77,Z 1155.625,A -85,B 0,C 180,E1 10724.922,E2 10724.922} C_VEL
LIN {X 0,Y 320.222,Z 1160.429,A -85,B 0,C 180,E1 10721.345,E2 10721.345} C_VEL
LIN {X 0,Y 319.961,Z 1164.274,A -85,B 0,C 180,E1 10717.361,E2 10717.361} C_VEL
LIN {X 0,Y 319.947,Z 1166.226,A -85,B 0,C 180,E1 10713.942,E2 10713.942} C_VEL
LIN {X 0,Y 319.941,Z 1167.042,A -85,B 0,C 180,E1 10710.537,E2 10710.537} C_VEL
LIN {X 0,Y 319.931,Z 1166.513,A -85,B 0,C 180,E1 10706.775,E2 10706.775} C_VEL
LIN {X 0,Y 319.968,Z 1164.756,A -85,B 0,C 180,E1 10703.361,E2 10703.361} C_VEL
LIN {X 0,Y 320.123,Z 1161.51,A -85,B 0,C 180,E1 10699.563,E2 10699.563} C_VEL
LIN {X 0,Y 320.637,Z 1156.591,A -85,B 0,C 180,E1 10695.738,E2 10695.738} C_VEL
LIN {X 0,Y 321.672,Z 1150.255,A -85,B 0,C 180,E1 10691.891,E2 10691.891} C_VEL
LIN {X 0,Y 323.398,Z 1142.1,A -85,B 0,C 180,E1 10688.031,E2 10688.031} C_VEL
LIN {X 0,Y 325.968,Z 1132.294,A -85,B 0,C 180,E1 10684.179,E2 10684.179} C_VEL
LIN {X 0,Y 329.279,Z 1121.035,A -85,B 0,C 180,E1 10680.533,E2 10680.533} C_VEL
LIN {X 0,Y 333.526,Z 1107.831,A -85,B 0,C 180,E1 10676.934,E2 10676.934} C_VEL
LIN {X 0,Y 338.195,Z 1094.043,A -85,B 0,C 180,E1 10673.751,E2 10673.751} C_VEL
LIN {X 0,Y 343.442,Z 1078.63,A -85,B 0,C 180,E1 10670.75,E2 10670.75} C_VEL
LIN {X 0,Y 349.225,Z 1061.67,A -85,B 0,C 180,E1 10667.936,E2 10667.936} C_VEL
LIN {X 0,Y 354.825,Z 1044.524,A -85,B 0,C 180,E1 10665.553,E2 10665.553} C_VEL
LIN {X 0,Y 360.953,Z 1024.802,A -85,B 0,C 180,E1 10663.237,E2 10663.237} C_VEL
LIN {X 0,Y 366.419,Z 1005.829,A -85,B 0,C 180,E1 10661.375,E2 10661.375} C_VEL
LIN {X 0,Y 371.718,Z 985.345,A -85,B 0,C 180,E1 10659.709,E2 10659.709} C_VEL
LIN {X 0,Y 376.562,Z 964.515,A -85,B 0,C 180,E1 10658.314,E2 10658.314} C_VEL
LIN {X 0,Y 380.824,Z 942.477,A -85,B 0,C 180,E1 10657.147,E2 10657.147} C_VEL
LIN {X 0,Y 384.613,Z 918.573,A -85,B 0,C 180,E1 10656.169,E2 10656.169} C_VEL
LIN {X 0,Y 387.332,Z 895.93,A -85,B 0,C 180,E1 10655.497,E2 10655.497} C_VEL
LIN {X 0,Y 389.851,Z 857.581,A -85,B 0,C 180,E1 10654.679,E2 10654.679} C_VEL
LIN {X 0,Y 402.08,Z 650.958,A -85,B 0,C 180,E1 10650.52,E2 10650.52} C_VEL
LIN {X 0,Y 402.182,Z 647.676,A -85,B 0,C 180,E1 10650.433,E2 10650.433} C_VEL
LIN {X 0,Y 393.869,Z 634.599,A -85,B 0,C 180,E1 10648.051,E2 10648.051} C_VEL
LIN {X 0,Y 385.573,Z 622.369,A -85,B 0,C 180,E1 10645.414,E2 10645.414} C_VEL
LIN {X 0,Y 378.007,Z 612.015,A -85,B 0,C 180,E1 10642.717,E2 10642.717} C_VEL
LIN {X 0,Y 371.14,Z 603.014,A -85,B 0,C 180,E1 10639.925,E2 10639.925} C_VEL
LIN {X 0,Y 366.341,Z 597.205,A -85,B 0,C 180,E1 10637.717,E2 10637.717} C_VEL
LIN {X 0,Y 362.164,Z 592.136,A -85,B 0,C 180,E1 10635.533,E2 10635.533} C_VEL
LIN {X 0,Y 357.375,Z 586.557,A -85,B 0,C 180,E1 10632.604,E2 10632.604} C_VEL
LIN {X 0,Y 352.152,Z 580.712,A -85,B 0,C 180,E1 10628.49,E2 10628.49} C_VEL
LIN {X 0,Y 347.035,Z 575.883,A -85,B 0,C 180,E1 10621.485,E2 10621.485} C_VEL
LIN {X 0,Y 346.256,Z 575.133,A -85,B 0,C 180,E1 10618.014,E2 10618.014} C_VEL
LIN {X 0,Y 346.561,Z 576.317,A -85,B 0,C 180,E1 10614.37,E2 10614.37} C_VEL
LIN {X 0,Y 349.895,Z 580.386,A -85,B 0,C 180,E1 10608.377,E2 10608.377} C_VEL
LIN {X 0,Y 353.343,Z 585.059,A -85,B 0,C 180,E1 10604.91,E2 10604.91} C_VEL
LIN {X 0,Y 354.522,Z 586.461,A -85,B 0,C 180,E1 10603.955,E2 10603.955} C_VEL
LIN {X 0,Y 358.639,Z 591.957,A -85,B 0,C 180,E1 10601.047,E2 10601.047} C_VEL
LIN {X 0,Y 362.701,Z 597.317,A -85,B 0,C 180,E1 10598.661,E2 10598.661} C_VEL
LIN {X 0,Y 367.75,Z 604.196,A -85,B 0,C 180,E1 10596.102,E2 10596.102} C_VEL
LIN {X 0,Y 374.018,Z 612.989,A -85,B 0,C 180,E1 10593.356,E2 10593.356} C_VEL
LIN {X 0,Y 380.388,Z 622.357,A -85,B 0,C 180,E1 10590.904,E2 10590.904} C_VEL
LIN {X 0,Y 387.425,Z 633.064,A -85,B 0,C 180,E1 10588.492,E2 10588.492} C_VEL
LIN {X 0,Y 395.529,Z 646.335,A -85,B 0,C 180,E1 10585.992,E2 10585.992} C_VEL
LIN {X 0,Y 399.437,Z 653.417,A -85,B 0,C 180,E1 10584.861,E2 10584.861} C_VEL
LIN {X 0,Y 387.467,Z 883.912,A -85,B 0,C 180,E1 10580.503,E2 10580.503} C_VEL
LIN {X 0,Y 385.653,Z 906.44,A -85,B 0,C 180,E1 10579.991,E2 10579.991} C_VEL
LIN {X 0,Y 382.703,Z 929.259,A -85,B 0,C 180,E1 10579.251,E2 10579.251} C_VEL
LIN {X 0,Y 379.228,Z 949.967,A -85,B 0,C 180,E1 10578.336,E2 10578.336} C_VEL
LIN {X 0,Y 374.927,Z 970.232,A -85,B 0,C 180,E1 10577.17,E2 10577.17} C_VEL
LIN {X 0,Y 369.732,Z 991.144,A -85,B 0,C 180,E1 10575.667,E2 10575.667} C_VEL
LIN {X 0,Y 364.328,Z 1010.271,A -85,B 0,C 180,E1 10573.974,E2 10573.974} C_VEL
LIN {X 0,Y 358.576,Z 1028.344,A -85,B 0,C 180,E1 10572.007,E2 10572.007} C_VEL
LIN {X 0,Y 352.451,Z 1046.197,A -85,B 0,C 180,E1 10569.665,E2 10569.665} C_VEL
LIN {X 0,Y 346.871,Z 1061.577,A -85,B 0,C 180,E1 10567.253,E2 10567.253} C_VEL
LIN {X 0,Y 341.203,Z 1076.411,A -85,B 0,C 180,E1 10564.442,E2 10564.442} C_VEL
LIN {X 0,Y 335.754,Z 1090.602,A -85,B 0,C 180,E1 10561.209,E2 10561.209} C_VEL
LIN {X 0,Y 331.218,Z 1102.674,A -85,B 0,C 180,E1 10557.898,E2 10557.898} C_VEL
LIN {X 0,Y 327.382,Z 1113.22,A -85,B 0,C 180,E1 10554.35,E2 10554.35} C_VEL
LIN {X 0,Y 324.366,Z 1122.382,A -85,B 0,C 180,E1 10550.573,E2 10550.573} C_VEL
LIN {X 0,Y 322.29,Z 1129.813,A -85,B 0,C 180,E1 10546.769,E2 10546.769} C_VEL
LIN {X 0,Y 320.959,Z 1135.65,A -85,B 0,C 180,E1 10542.821,E2 10542.821} C_VEL
LIN {X 0,Y 320.288,Z 1139.952,A -85,B 0,C 180,E1 10538.799,E2 10538.799} C_VEL
LIN {X 0,Y 320.029,Z 1142.464,A -85,B 0,C 180,E1 10535.198,E2 10535.198} C_VEL
LIN {X 0,Y 319.971,Z 1143.664,A -85,B 0,C 180,E1 10531.432,E2 10531.432} C_VEL
LIN {X 0,Y 319.975,Z 1143.612,A -85,B 0,C 180,E1 10528.03,E2 10528.03} C_VEL
LIN {X 0,Y 320.013,Z 1142.918,A -85,B 0,C 180,E1 10525.736,E2 10525.736} C_VEL
LIN {X 0,Y 319.07,Z 1142.383,A -85,B 0,C 180,E1 10524.358,E2 10524.358} C_VEL
LIN {X 0,Y 314.773,Z 1141.024,A -85,B 0,C 180,E1 10521.851,E2 10521.851} C_VEL
LIN {X 0,Y 312.62,Z 1139.591,A -85,B 0,C 180,E1 10520.068,E2 10520.068} C_VEL
LIN {X 0,Y 312.502,Z 1138.983,A -85,B 0,C 180,E1 10519.463,E2 10519.463} C_VEL
LIN {X 0,Y 313.398,Z 1134.448,A -85,B 0,C 180,E1 10515.59,E2 10515.59} C_VEL
LIN {X 0,Y 315.096,Z 1127.966,A -85,B 0,C 180,E1 10511.499,E2 10511.499} C_VEL
LIN {X 0,Y 317.625,Z 1120.114,A -85,B 0,C 180,E1 10507.61,E2 10507.61} C_VEL
LIN {X 0,Y 320.968,Z 1110.827,A -85,B 0,C 180,E1 10503.945,E2 10503.945} C_VEL
LIN {X 0,Y 325.295,Z 1099.669,A -85,B 0,C 180,E1 10500.339,E2 10500.339} C_VEL
LIN {X 0,Y 330.089,Z 1087.884,A -85,B 0,C 180,E1 10497.166,E2 10497.166} C_VEL
LIN {X 0,Y 335.693,Z 1073.901,A -85,B 0,C 180,E1 10494.072,E2 10494.072} C_VEL
LIN {X 0,Y 341.766,Z 1058.505,A -85,B 0,C 180,E1 10491.239,E2 10491.239} C_VEL
LIN {X 0,Y 347.739,Z 1042.79,A -85,B 0,C 180,E1 10488.818,E2 10488.818} C_VEL
LIN {X 0,Y 353.786,Z 1025.51,A -85,B 0,C 180,E1 10486.626,E2 10486.626} C_VEL
LIN {X 0,Y 359.839,Z 1006.786,A -85,B 0,C 180,E1 10484.657,E2 10484.657} C_VEL
LIN {X 0,Y 365.26,Z 988.119,A -85,B 0,C 180,E1 10483.039,E2 10483.039} C_VEL
LIN {X 0,Y 370.172,Z 968.516,A -85,B 0,C 180,E1 10481.67,E2 10481.67} C_VEL
LIN {X 0,Y 374.537,Z 948.137,A -85,B 0,C 180,E1 10480.521,E2 10480.521} C_VEL
LIN {X 0,Y 378.142,Z 927.161,A -85,B 0,C 180,E1 10479.614,E2 10479.614} C_VEL
LIN {X 0,Y 381.024,Z 904.883,A -85,B 0,C 180,E1 10478.917,E2 10478.917} C_VEL
LIN {X 0,Y 382.859,Z 881.575,A -85,B 0,C 180,E1 10478.398,E2 10478.398} C_VEL
LIN {X 0,Y 390.11,Z 743.316,A -85,B 0,C 180,E1 10475.759,E2 10475.759} C_VEL
LIN {X 0,Y 384.62,Z 752.682,A -85,B 0,C 180,E1 10474.799,E2 10474.799} C_VEL
LIN {X 0,Y 379.833,Z 771.816,A -85,B 0,C 180,E1 10474.287,E2 10474.287} C_VEL
LIN {X 0,Y 375.983,Z 783.719,A -85,B 0,C 180,E1 10473.743,E2 10473.743} C_VEL
LIN {X 0,Y 374.408,Z 788.217,A -85,B 0,C 180,E1 10473.502,E2 10473.502} C_VEL
LIN {X 0,Y 368.646,Z 814.243,A -85,B 0,C 180,E1 10472.932,E2 10472.932} C_VEL
LIN {X 0,Y 364.676,Z 828.618,A -85,B 0,C 180,E1 10472.394,E2 10472.394} C_VEL
LIN {X 0,Y 361.308,Z 838.185,A -85,B 0,C 180,E1 10471.824,E2 10471.824} C_VEL
LIN {X 0,Y 355.466,Z 864.975,A -85,B 0,C 180,E1 10471.187,E2 10471.187} C_VEL
LIN {X 0,Y 351.682,Z 878.847,A -85,B 0,C 180,E1 10470.615,E2 10470.615} C_VEL
LIN {X 0,Y 348.533,Z 887.635,A -85,B 0,C 180,E1 10470.04,E2 10470.04} C_VEL
LIN {X 0,Y 344.142,Z 904.335,A -85,B 0,C 180,E1 10469.61,E2 10469.61} C_VEL
LIN {X 0,Y 340.772,Z 913.153,A -85,B 0,C 180,E1 10469.172,E2 10469.172} C_VEL
LIN {X 0,Y 337.648,Z 918.712,A -85,B 0,C 180,E1 10468.619,E2 10468.619} C_VEL
LIN {X 0,Y 335.724,Z 921.564,A -85,B 0,C 180,E1 10468.216,E2 10468.216} C_VEL
LIN {X 0,Y 331.492,Z 930.645,A -85,B 0,C 180,E1 10467.678,E2 10467.678} C_VEL
LIN {X 0,Y 328.575,Z 935.332,A -85,B 0,C 180,E1 10467.159,E2 10467.159} C_VEL
LIN {X 0,Y 325.981,Z 938.653,A -85,B 0,C 180,E1 10466.408,E2 10466.408} C_VEL
LIN {X 0,Y 325.471,Z 941.885,A -85,B 0,C 180,E1 10466.06,E2 10466.06} C_VEL
LIN {X 0,Y 324.036,Z 959.43,A -85,B 0,C 180,E1 10464.618,E2 10464.618} C_VEL
LIN {X 0,Y 322.458,Z 975.67,A -85,B 0,C 180,E1 10462.902,E2 10462.902} C_VEL
LIN {X 0,Y 320.803,Z 990.877,A -85,B 0,C 180,E1 10460.908,E2 10460.908} C_VEL
LIN {X 0,Y 319.238,Z 1004.19,A -85,B 0,C 180,E1 10458.738,E2 10458.738} C_VEL
LIN {X 0,Y 317.775,Z 1016.565,A -85,B 0,C 180,E1 10456.263,E2 10456.263} C_VEL
LIN {X 0,Y 316.609,Z 1026.892,A -85,B 0,C 180,E1 10453.701,E2 10453.701} C_VEL
LIN {X 0,Y 315.69,Z 1035.754,A -85,B 0,C 180,E1 10450.935,E2 10450.935} C_VEL
LIN {X 0,Y 315.098,Z 1043.024,A -85,B 0,C 180,E1 10448.026,E2 10448.026} C_VEL
LIN {X 0,Y 314.812,Z 1048.334,A -85,B 0,C 180,E1 10445.103,E2 10445.103} C_VEL
LIN {X 0,Y 314.806,Z 1052.057,A -85,B 0,C 180,E1 10442.003,E2 10442.003} C_VEL
LIN {X 0,Y 315.044,Z 1053.872,A -85,B 0,C 180,E1 10439.091,E2 10439.091} C_VEL
LIN {X 0,Y 315.468,Z 1053.954,A -85,B 0,C 180,E1 10436.184,E2 10436.184} C_VEL
LIN {X 0,Y 316.222,Z 1052.212,A -85,B 0,C 180,E1 10433.1,E2 10433.1} C_VEL
LIN {X 0,Y 317.277,Z 1048.792,A -85,B 0,C 180,E1 10430.203,E2 10430.203} C_VEL
LIN {X 0,Y 318.681,Z 1043.372,A -85,B 0,C 180,E1 10427.314,E2 10427.314} C_VEL
LIN {X 0,Y 320.357,Z 1036.365,A -85,B 0,C 180,E1 10424.616,E2 10424.616} C_VEL
LIN {X 0,Y 322.238,Z 1027.828,A -85,B 0,C 180,E1 10422.111,E2 10422.111} C_VEL
LIN {X 0,Y 324.234,Z 1017.701,A -85,B 0,C 180,E1 10419.796,E2 10419.796} C_VEL
LIN {X 0,Y 326.311,Z 1006.139,A -85,B 0,C 180,E1 10417.67,E2 10417.67} C_VEL
LIN {X 0,Y 328.339,Z 992.849,A -85,B 0,C 180,E1 10415.727,E2 10415.727} C_VEL
LIN {X 0,Y 330.165,Z 978.644,A -85,B 0,C 180,E1 10414.06,E2 10414.06} C_VEL
LIN {X 0,Y 332.232,Z 961.088,A -85,B 0,C 180,E1 10412.39,E2 10412.39} C_VEL
LIN {X 0,Y 335.543,Z 957.701,A -85,B 0,C 180,E1 10411.72,E2 10411.72} C_VEL
LIN {X 0,Y 339.152,Z 953.05,A -85,B 0,C 180,E1 10411.28,E2 10411.28} C_VEL
LIN {X 0,Y 341.097,Z 950.244,A -85,B 0,C 180,E1 10411.076,E2 10411.076} C_VEL
LIN {X 0,Y 344.968,Z 945.972,A -85,B 0,C 180,E1 10410.48,E2 10410.48} C_VEL
LIN {X 0,Y 348.785,Z 940.202,A -85,B 0,C 180,E1 10410.08,E2 10410.08} C_VEL
LIN {X 0,Y 351.479,Z 935.385,A -85,B 0,C 180,E1 10409.86,E2 10409.86} C_VEL
LIN {X 0,Y 355.717,Z 929.306,A -85,B 0,C 180,E1 10409.316,E2 10409.316} C_VEL
LIN {X 0,Y 360.064,Z 920.719,A -85,B 0,C 180,E1 10408.949,E2 10408.949} C_VEL
LIN {X 0,Y 363.476,Z 912.263,A -85,B 0,C 180,E1 10408.721,E2 10408.721} C_VEL
LIN {X 0,Y 367.592,Z 904.282,A -85,B 0,C 180,E1 10408.243,E2 10408.243} C_VEL
LIN {X 0,Y 372.089,Z 892.174,A -85,B 0,C 180,E1 10407.845,E2 10407.845} C_VEL
LIN {X 0,Y 377.522,Z 872.403,A -85,B 0,C 180,E1 10407.396,E2 10407.396} C_VEL
LIN {X 0,Y 381.988,Z 860.674,A -85,B 0,C 180,E1 10406.835,E2 10406.835} C_VEL
LIN {X 0,Y 385.654,Z 848.885,A -85,B 0,C 180,E1 10406.459,E2 10406.459} C_VEL
LIN {X 0,Y 382.631,Z 895.098,A -85,B 0,C 180,E1 10405.483,E2 10405.483} C_VEL
LIN {X 0,Y 379.826,Z 917.952,A -85,B 0,C 180,E1 10404.807,E2 10404.807} C_VEL
LIN {X 0,Y 376.058,Z 941.242,A -85,B 0,C 180,E1 10403.868,E2 10403.868} C_VEL
LIN {X 0,Y 371.923,Z 962.07,A -85,B 0,C 180,E1 10402.781,E2 10402.781} C_VEL
LIN {X 0,Y 366.775,Z 983.809,A -85,B 0,C 180,E1 10401.355,E2 10401.355} C_VEL
LIN {X 0,Y 361.32,Z 1004.35,A -85,B 0,C 180,E1 10399.706,E2 10399.706} C_VEL
LIN {X 0,Y 355.542,Z 1023.636,A -85,B 0,C 180,E1 10397.818,E2 10397.818} C_VEL
LIN {X 0,Y 348.953,Z 1044.077,A -85,B 0,C 180,E1 10395.413,E2 10395.413} C_VEL
LIN {X 0,Y 343.013,Z 1061.448,A -85,B 0,C 180,E1 10392.976,E2 10392.976} C_VEL
LIN {X 0,Y 337.082,Z 1077.987,A -85,B 0,C 180,E1 10390.206,E2 10390.206} C_VEL
LIN {X 0,Y 331.458,Z 1093.702,A -85,B 0,C 180,E1 10387.108,E2 10387.108} C_VEL
LIN {X 0,Y 326.507,Z 1107.489,A -85,B 0,C 180,E1 10383.872,E2 10383.872} C_VEL
LIN {X 0,Y 321.797,Z 1121.297,A -85,B 0,C 180,E1 10380.016,E2 10380.016} C_VEL
LIN {X 0,Y 318.312,Z 1132.498,A -85,B 0,C 180,E1 10376.289,E2 10376.289} C_VEL
LIN {X 0,Y 315.573,Z 1142.29,A -85,B 0,C 180,E1 10372.308,E2 10372.308} C_VEL
LIN {X 0,Y 313.694,Z 1150.588,A -85,B 0,C 180,E1 10368.202,E2 10368.202} C_VEL
LIN {X 0,Y 312.668,Z 1156.554,A -85,B 0,C 180,E1 10364.444,E2 10364.444} C_VEL
LIN {X 0,Y 312.112,Z 1161.559,A -85,B 0,C 180,E1 10360.335,E2 10360.335} C_VEL
LIN {X 0,Y 311.966,Z 1164.463,A -85,B 0,C 180,E1 10356.811,E2 10356.811} C_VEL
LIN {X 0,Y 311.938,Z 1166.15,A -85,B 0,C 180,E1 10353.492,E2 10353.492} C_VEL
LIN {X 0,Y 311.954,Z 1166.796,A -85,B 0,C 180,E1 10349.798,E2 10349.798} C_VEL
LIN {X 0,Y 311.949,Z 1166.004,A -85,B 0,C 180,E1 10346.141,E2 10346.141} C_VEL
LIN {X 0,Y 311.96,Z 1164.218,A -85,B 0,C 180,E1 10342.819,E2 10342.819} C_VEL
LIN {X 0,Y 312.194,Z 1160.775,A -85,B 0,C 180,E1 10338.921,E2 10338.921} C_VEL
LIN {X 0,Y 312.742,Z 1156.011,A -85,B 0,C 180,E1 10335.181,E2 10335.181} C_VEL
LIN {X 0,Y 313.906,Z 1149.575,A -85,B 0,C 180,E1 10331.234,E2 10331.234} C_VEL
LIN {X 0,Y 315.819,Z 1141.345,A -85,B 0,C 180,E1 10327.279,E2 10327.279} C_VEL
LIN {X 0,Y 318.772,Z 1130.875,A -85,B 0,C 180,E1 10323.149,E2 10323.149} C_VEL
LIN {X 0,Y 322.201,Z 1120.086,A -85,B 0,C 180,E1 10319.614,E2 10319.614} C_VEL
LIN {X 0,Y 326.752,Z 1106.733,A -85,B 0,C 180,E1 10315.946,E2 10315.946} C_VEL
LIN {X 0,Y 331.756,Z 1092.866,A -85,B 0,C 180,E1 10312.715,E2 10312.715} C_VEL
LIN {X 0,Y 337.203,Z 1077.582,A -85,B 0,C 180,E1 10309.729,E2 10309.729} C_VEL
LIN {X 0,Y 343.25,Z 1060.658,A -85,B 0,C 180,E1 10306.915,E2 10306.915} C_VEL
LIN {X 0,Y 348.929,Z 1044.039,A -85,B 0,C 180,E1 10304.591,E2 10304.591} C_VEL
LIN {X 0,Y 355.53,Z 1023.531,A -85,B 0,C 180,E1 10302.179,E2 10302.179} C_VEL
LIN {X 0,Y 361.491,Z 1003.612,A -85,B 0,C 180,E1 10300.235,E2 10300.235} C_VEL
LIN {X 0,Y 366.841,Z 983.354,A -85,B 0,C 180,E1 10298.62,E2 10298.62} C_VEL
LIN {X 0,Y 372.063,Z 961.132,A -85,B 0,C 180,E1 10297.175,E2 10297.175} C_VEL
LIN {X 0,Y 376.175,Z 940.327,A -85,B 0,C 180,E1 10296.097,E2 10296.097} C_VEL
LIN {X 0,Y 379.862,Z 917.253,A -85,B 0,C 180,E1 10295.177,E2 10295.177} C_VEL
LIN {X 0,Y 382.666,Z 894.132,A -85,B 0,C 180,E1 10294.501,E2 10294.501} C_VEL
LIN {X 0,Y 387.051,Z 824.646,A -85,B 0,C 180,E1 10293.054,E2 10293.054} C_VEL
LIN {X 0,Y 397.677,Z 651.929,A -85,B 0,C 180,E1 10289.565,E2 10289.565} C_VEL
LIN {X 0,Y 388.537,Z 637.538,A -85,B 0,C 180,E1 10286.807,E2 10286.807} C_VEL
LIN {X 0,Y 379.81,Z 624.734,A -85,B 0,C 180,E1 10283.834,E2 10283.834} C_VEL
LIN {X 0,Y 372.412,Z 614.728,A -85,B 0,C 180,E1 10280.962,E2 10280.962} C_VEL
LIN {X 0,Y 367.508,Z 608.435,A -85,B 0,C 180,E1 10278.807,E2 10278.807} C_VEL
LIN {X 0,Y 364.283,Z 604.397,A -85,B 0,C 180,E1 10277.243,E2 10277.243} C_VEL
LIN {X 0,Y 360.351,Z 599.548,A -85,B 0,C 180,E1 10275.118,E2 10275.118} C_VEL
LIN {X 0,Y 355.923,Z 594.249,A -85,B 0,C 180,E1 10272.327,E2 10272.327} C_VEL
LIN {X 0,Y 350.822,Z 588.452,A -85,B 0,C 180,E1 10268.192,E2 10268.192} C_VEL
LIN {X 0,Y 345.992,Z 583.768,A -85,B 0,C 180,E1 10261.324,E2 10261.324} C_VEL
LIN {X 0,Y 345.281,Z 583.075,A -85,B 0,C 180,E1 10258.008,E2 10258.008} C_VEL
LIN {X 0,Y 345.586,Z 584.295,A -85,B 0,C 180,E1 10254.354,E2 10254.354} C_VEL
LIN {X 0,Y 348.727,Z 588.214,A -85,B 0,C 180,E1 10248.589,E2 10248.589} C_VEL
LIN {X 0,Y 352.201,Z 592.953,A -85,B 0,C 180,E1 10245.028,E2 10245.028} C_VEL
LIN {X 0,Y 353.444,Z 594.693,A -85,B 0,C 180,E1 10243.989,E2 10243.989} C_VEL
LIN {X 0,Y 357.189,Z 599.725,A -85,B 0,C 180,E1 10241.306,E2 10241.306} C_VEL
LIN {X 0,Y 361.045,Z 604.92,A -85,B 0,C 180,E1 10238.983,E2 10238.983} C_VEL
LIN {X 0,Y 365.929,Z 611.693,A -85,B 0,C 180,E1 10236.446,E2 10236.446} C_VEL
LIN {X 0,Y 372.089,Z 620.548,A -85,B 0,C 180,E1 10233.68,E2 10233.68} C_VEL
LIN {X 0,Y 378.083,Z 629.545,A -85,B 0,C 180,E1 10231.315,E2 10231.315} C_VEL
LIN {X 0,Y 385.001,Z 640.356,A -85,B 0,C 180,E1 10228.881,E2 10228.881} C_VEL
LIN {X 0,Y 392.544,Z 652.937,A -85,B 0,C 180,E1 10226.489,E2 10226.489} C_VEL
LIN {X 0,Y 394.943,Z 657.475,A -85,B 0,C 180,E1 10225.764,E2 10225.764} C_VEL
LIN {X 0,Y 382.248,Z 890.185,A -85,B 0,C 180,E1 10221.328,E2 10221.328} C_VEL
LIN {X 0,Y 380.134,Z 912.452,A -85,B 0,C 180,E1 10220.778,E2 10220.778} C_VEL
LIN {X 0,Y 377.19,Z 932.827,A -85,B 0,C 180,E1 10220.063,E2 10220.063} C_VEL
LIN {X 0,Y 373.257,Z 954.224,A -85,B 0,C 180,E1 10219.061,E2 10219.061} C_VEL
LIN {X 0,Y 369.031,Z 973.182,A -85,B 0,C 180,E1 10217.935,E2 10217.935} C_VEL
LIN {X 0,Y 363.925,Z 992.612,A -85,B 0,C 180,E1 10216.496,E2 10216.496} C_VEL
LIN {X 0,Y 358.34,Z 1011.501,A -85,B 0,C 180,E1 10214.793,E2 10214.793} C_VEL
LIN {X 0,Y 352.613,Z 1028.805,A -85,B 0,C 180,E1 10212.886,E2 10212.886} C_VEL
LIN {X 0,Y 346.243,Z 1046.612,A -85,B 0,C 180,E1 10210.522,E2 10210.522} C_VEL
LIN {X 0,Y 340.43,Z 1061.975,A -85,B 0,C 180,E1 10208.082,E2 10208.082} C_VEL
LIN {X 0,Y 334.499,Z 1076.781,A -85,B 0,C 180,E1 10205.233,E2 10205.233} C_VEL
LIN {X 0,Y 328.784,Z 1090.95,A -85,B 0,C 180,E1 10201.948,E2 10201.948} C_VEL
LIN {X 0,Y 323.998,Z 1103.006,A -85,B 0,C 180,E1 10198.577,E2 10198.577} C_VEL
LIN {X 0,Y 319.936,Z 1113.548,A -85,B 0,C 180,E1 10194.955,E2 10194.955} C_VEL
LIN {X 0,Y 316.721,Z 1122.698,A -85,B 0,C 180,E1 10191.093,E2 10191.093} C_VEL
LIN {X 0,Y 314.499,Z 1130.119,A -85,B 0,C 180,E1 10187.198,E2 10187.198} C_VEL
LIN {X 0,Y 313.091,Z 1135.768,A -85,B 0,C 180,E1 10183.293,E2 10183.293} C_VEL
LIN {X 0,Y 312.346,Z 1140.099,A -85,B 0,C 180,E1 10179.21,E2 10179.21} C_VEL
LIN {X 0,Y 312.051,Z 1142.65,A -85,B 0,C 180,E1 10175.516,E2 10175.516} C_VEL
LIN {X 0,Y 311.976,Z 1143.934,A -85,B 0,C 180,E1 10171.653,E2 10171.653} C_VEL
LIN {X 0,Y 311.979,Z 1143.924,A -85,B 0,C 180,E1 10168.163,E2 10168.163} C_VEL
LIN {X 0,Y 312.058,Z 1142.6,A -85,B 0,C 180,E1 10164.3,E2 10164.3} C_VEL
LIN {X 0,Y 312.358,Z 1140.028,A -85,B 0,C 180,E1 10160.604,E2 10160.604} C_VEL
LIN {X 0,Y 312.502,Z 1138.983,A -85,B 0,C 180,E1 10159.463,E2 10159.463} C_VEL
LIN {X 0,Y 311.753,Z 1137.606,A -85,B 0,C 180,E1 10158.07,E2 10158.07} C_VEL
LIN {X 0,Y 306.504,Z 1133.341,A -85,B 0,C 180,E1 10154.218,E2 10154.218} C_VEL
LIN {X 0,Y 306.324,Z 1131.723,A -85,B 0,C 180,E1 10153.11,E2 10153.11} C_VEL
LIN {X 0,Y 308.778,Z 1123.984,A -85,B 0,C 180,E1 10148.736,E2 10148.736} C_VEL
LIN {X 0,Y 312.083,Z 1115.106,A -85,B 0,C 180,E1 10144.779,E2 10144.779} C_VEL
LIN {X 0,Y 316.247,Z 1104.711,A -85,B 0,C 180,E1 10141.07,E2 10141.07} C_VEL
LIN {X 0,Y 321.455,Z 1092.323,A -85,B 0,C 180,E1 10137.451,E2 10137.451} C_VEL
LIN {X 0,Y 327.066,Z 1079.189,A -85,B 0,C 180,E1 10134.275,E2 10134.275} C_VEL
LIN {X 0,Y 333.139,Z 1064.611,A -85,B 0,C 180,E1 10131.371,E2 10131.371} C_VEL
LIN {X 0,Y 339.541,Z 1048.625,A -85,B 0,C 180,E1 10128.729,E2 10128.729} C_VEL
LIN {X 0,Y 345.87,Z 1031.935,A -85,B 0,C 180,E1 10126.426,E2 10126.426} C_VEL
LIN {X 0,Y 352.002,Z 1014.118,A -85,B 0,C 180,E1 10124.407,E2 10124.407} C_VEL
LIN {X 0,Y 358.016,Z 994.897,A -85,B 0,C 180,E1 10122.617,E2 10122.617} C_VEL
LIN {X 0,Y 363.28,Z 975.929,A -85,B 0,C 180,E1 10121.17,E2 10121.17} C_VEL
LIN {X 0,Y 367.9,Z 956.192,A -85,B 0,C 180,E1 10119.967,E2 10119.967} C_VEL
LIN {X 0,Y 371.984,Z 935.383,A -85,B 0,C 180,E1 10118.962,E2 10118.962} C_VEL
LIN {X 0,Y 375.056,Z 915.157,A -85,B 0,C 180,E1 10118.231,E2 10118.231} C_VEL
LIN {X 0,Y 377.504,Z 891.82,A -85,B 0,C 180,E1 10117.629,E2 10117.629} C_VEL
LIN {X 0,Y 384.087,Z 772.764,A -85,B 0,C 180,E1 10115.325,E2 10115.325} C_VEL
LIN {X 0,Y 379.973,Z 785.759,A -85,B 0,C 180,E1 10114.783,E2 10114.783} C_VEL
LIN {X 0,Y 378.083,Z 791.117,A -85,B 0,C 180,E1 10114.508,E2 10114.508} C_VEL
LIN {X 0,Y 372.363,Z 816.578,A -85,B 0,C 180,E1 10113.966,E2 10113.966} C_VEL
LIN {X 0,Y 368.21,Z 831.409,A -85,B 0,C 180,E1 10113.429,E2 10113.429} C_VEL
LIN {X 0,Y 364.713,Z 841.39,A -85,B 0,C 180,E1 10112.87,E2 10112.87} C_VEL
LIN {X 0,Y 359.174,Z 866.59,A -85,B 0,C 180,E1 10112.298,E2 10112.298} C_VEL
LIN {X 0,Y 355.172,Z 881.187,A -85,B 0,C 180,E1 10111.729,E2 10111.729} C_VEL
LIN {X 0,Y 351.568,Z 891.14,A -85,B 0,C 180,E1 10111.129,E2 10111.129} C_VEL
LIN {X 0,Y 347.34,Z 906.657,A -85,B 0,C 180,E1 10110.764,E2 10110.764} C_VEL
LIN {X 0,Y 343.462,Z 916.441,A -85,B 0,C 180,E1 10110.313,E2 10110.313} C_VEL
LIN {X 0,Y 339.823,Z 923.068,A -85,B 0,C 180,E1 10109.721,E2 10109.721} C_VEL
LIN {X 0,Y 337.53,Z 926.431,A -85,B 0,C 180,E1 10109.309,E2 10109.309} C_VEL
LIN {X 0,Y 333.069,Z 935.338,A -85,B 0,C 180,E1 10108.768,E2 10108.768} C_VEL
LIN {X 0,Y 329.75,Z 940.376,A -85,B 0,C 180,E1 10108.231,E2 10108.231} C_VEL
LIN {X 0,Y 326.571,Z 943.814,A -85,B 0,C 180,E1 10107.537,E2 10107.537} C_VEL
LIN {X 0,Y 325.936,Z 944.51,A -85,B 0,C 180,E1 10107.397,E2 10107.397} C_VEL
LIN {X 0,Y 321.792,Z 951.043,A -85,B 0,C 180,E1 10106.779,E2 10106.779} C_VEL
LIN {X 0,Y 319.106,Z 954.157,A -85,B 0,C 180,E1 10106.219,E2 10106.219} C_VEL
LIN {X 0,Y 317.078,Z 956.141,A -85,B 0,C 180,E1 10105.546,E2 10105.546} C_VEL
LIN {X 0,Y 316.443,Z 960.18,A -85,B 0,C 180,E1 10105.05,E2 10105.05} C_VEL
LIN {X 0,Y 314.892,Z 975.777,A -85,B 0,C 180,E1 10103.385,E2 10103.385} C_VEL
LIN {X 0,Y 313.163,Z 991.223,A -85,B 0,C 180,E1 10101.345,E2 10101.345} C_VEL
LIN {X 0,Y 311.593,Z 1004.368,A -85,B 0,C 180,E1 10099.203,E2 10099.203} C_VEL
LIN {X 0,Y 310.057,Z 1016.929,A -85,B 0,C 180,E1 10096.679,E2 10096.679} C_VEL
LIN {X 0,Y 308.832,Z 1027.538,A -85,B 0,C 180,E1 10094.053,E2 10094.053} C_VEL
LIN {X 0,Y 307.864,Z 1036.538,A -85,B 0,C 180,E1 10091.237,E2 10091.237} C_VEL
LIN {X 0,Y 307.225,Z 1044.016,A -85,B 0,C 180,E1 10088.233,E2 10088.233} C_VEL
LIN {X 0,Y 306.928,Z 1049.527,A -85,B 0,C 180,E1 10085.234,E2 10085.234} C_VEL
LIN {X 0,Y 306.917,Z 1053.222,A -85,B 0,C 180,E1 10082.241,E2 10082.241} C_VEL
LIN {X 0,Y 307.158,Z 1055.266,A -85,B 0,C 180,E1 10079.254,E2 10079.254} C_VEL
LIN {X 0,Y 307.634,Z 1055.632,A -85,B 0,C 180,E1 10076.201,E2 10076.201} C_VEL
LIN {X 0,Y 308.414,Z 1054.123,A -85,B 0,C 180,E1 10073.111,E2 10073.111} C_VEL
LIN {X 0,Y 309.532,Z 1050.918,A -85,B 0,C 180,E1 10070.138,E2 10070.138} C_VEL
LIN {X 0,Y 310.934,Z 1046.21,A -85,B 0,C 180,E1 10067.37,E2 10067.37} C_VEL
LIN {X 0,Y 312.683,Z 1039.577,A -85,B 0,C 180,E1 10064.609,E2 10064.609} C_VEL
LIN {X 0,Y 314.641,Z 1031.46,A -85,B 0,C 180,E1 10062.047,E2 10062.047} C_VEL
LIN {X 0,Y 316.869,Z 1021.492,A -85,B 0,C 180,E1 10059.581,E2 10059.581} C_VEL
LIN {X 0,Y 319.227,Z 1009.4,A -85,B 0,C 180,E1 10057.244,E2 10057.244} C_VEL
LIN {X 0,Y 321.39,Z 996.774,A -85,B 0,C 180,E1 10055.29,E2 10055.29} C_VEL
LIN {X 0,Y 323.499,Z 982.092,A -85,B 0,C 180,E1 10053.474,E2 10053.474} C_VEL
LIN {X 0,Y 324.553,Z 974.803,A -85,B 0,C 180,E1 10052.676,E2 10052.676} C_VEL
LIN {X 0,Y 326.268,Z 973.133,A -85,B 0,C 180,E1 10052.238,E2 10052.238} C_VEL
LIN {X 0,Y 329.805,Z 969.903,A -85,B 0,C 180,E1 10051.677,E2 10051.677} C_VEL
LIN {X 0,Y 333.006,Z 966.179,A -85,B 0,C 180,E1 10051.289,E2 10051.289} C_VEL
LIN {X 0,Y 336.864,Z 962.71,A -85,B 0,C 180,E1 10050.677,E2 10050.677} C_VEL
LIN {X 0,Y 341.513,Z 956.736,A -85,B 0,C 180,E1 10050.152,E2 10050.152} C_VEL
LIN {X 0,Y 343.004,Z 954.978,A -85,B 0,C 180,E1 10049.97,E2 10049.97} C_VEL
LIN {X 0,Y 347.547,Z 949.876,A -85,B 0,C 180,E1 10049.389,E2 10049.389} C_VEL
LIN {X 0,Y 352.002,Z 943.011,A -85,B 0,C 180,E1 10048.966,E2 10048.966} C_VEL
LIN {X 0,Y 353.693,Z 940.031,A -85,B 0,C 180,E1 10048.848,E2 10048.848} C_VEL
LIN {X 0,Y 358.464,Z 933.357,A -85,B 0,C 180,E1 10048.301,E2 10048.301} C_VEL
LIN {X 0,Y 363.261,Z 924.278,A -85,B 0,C 180,E1 10047.924,E2 10047.924} C_VEL
LIN {X 0,Y 366.896,Z 915.65,A -85,B 0,C 180,E1 10047.692,E2 10047.692} C_VEL
LIN {X 0,Y 371.6,Z 906.555,A -85,B 0,C 180,E1 10047.215,E2 10047.215} C_VEL
LIN {X 0,Y 376.454,Z 893.559,A -85,B 0,C 180,E1 10046.83,E2 10046.83} C_VEL
LIN {X 0,Y 378.626,Z 886.042,A -85,B 0,C 180,E1 10046.665,E2 10046.665} C_VEL
LIN {X 0,Y 376.248,Z 909.388,A -85,B 0,C 180,E1 10046.063,E2 10046.063} C_VEL
LIN {X 0,Y 372.968,Z 930.87,A -85,B 0,C 180,E1 10045.295,E2 10045.295} C_VEL
LIN {X 0,Y 368.873,Z 952.748,A -85,B 0,C 180,E1 10044.274,E2 10044.274} C_VEL
LIN {X 0,Y 364.298,Z 972.903,A -85,B 0,C 180,E1 10043.079,E2 10043.079} C_VEL
LIN {X 0,Y 358.544,Z 994.927,A -85,B 0,C 180,E1 10041.465,E2 10041.465} C_VEL
LIN {X 0,Y 352.971,Z 1013.917,A -85,B 0,C 180,E1 10039.771,E2 10039.771} C_VEL
LIN {X 0,Y 346.734,Z 1033.138,A -85,B 0,C 180,E1 10037.702,E2 10037.702} C_VEL
LIN {X 0,Y 340.302,Z 1051.748,A -85,B 0,C 180,E1 10035.319,E2 10035.319} C_VEL
LIN {X 0,Y 334.084,Z 1068.645,A -85,B 0,C 180,E1 10032.712,E2 10032.712} C_VEL
LIN {X 0,Y 327.718,Z 1085.565,A -85,B 0,C 180,E1 10029.617,E2 10029.617} C_VEL
LIN {X 0,Y 322.347,Z 1099.719,A -85,B 0,C 180,E1 10026.548,E2 10026.548} C_VEL
LIN {X 0,Y 317.285,Z 1113.335,A -85,B 0,C 180,E1 10023.037,E2 10023.037} C_VEL
LIN {X 0,Y 312.951,Z 1125.712,A -85,B 0,C 180,E1 10019.264,E2 10019.264} C_VEL
LIN {X 0,Y 309.45,Z 1136.517,A -85,B 0,C 180,E1 10015.246,E2 10015.246} C_VEL
LIN {X 0,Y 306.786,Z 1146.299,A -85,B 0,C 180,E1 10010.809,E2 10010.809} C_VEL
LIN {X 0,Y 305.291,Z 1153.147,A -85,B 0,C 180,E1 10006.947,E2 10006.947} C_VEL
LIN {X 0,Y 304.374,Z 1158.989,A -85,B 0,C 180,E1 10002.677,E2 10002.677} C_VEL
LIN {X 0,Y 304.055,Z 1162.619,A -85,B 0,C 180,E1 9999.082,E2 9999.082} C_VEL
LIN {X 0,Y 303.953,Z 1165.35,A -85,B 0,C 180,E1 9994.906,E2 9994.906} C_VEL
LIN {X 0,Y 303.962,Z 1166.365,A -85,B 0,C 180,E1 9991.319,E2 9991.319} C_VEL
LIN {X 0,Y 303.964,Z 1166.267,A -85,B 0,C 180,E1 9987.926,E2 9987.926} C_VEL
LIN {X 0,Y 303.953,Z 1164.768,A -85,B 0,C 180,E1 9983.958,E2 9983.958} C_VEL
LIN {X 0,Y 304.074,Z 1162.105,A -85,B 0,C 180,E1 9980.346,E2 9980.346} C_VEL
LIN {X 0,Y 304.522,Z 1157.84,A -85,B 0,C 180,E1 9976.326,E2 9976.326} C_VEL
LIN {X 0,Y 305.546,Z 1151.763,A -85,B 0,C 180,E1 9972.222,E2 9972.222} C_VEL
LIN {X 0,Y 307.359,Z 1143.987,A -85,B 0,C 180,E1 9968.031,E2 9968.031} C_VEL
LIN {X 0,Y 309.879,Z 1135.063,A -85,B 0,C 180,E1 9964.177,E2 9964.177} C_VEL
LIN {X 0,Y 313.537,Z 1123.887,A -85,B 0,C 180,E1 9960.156,E2 9960.156} C_VEL
LIN {X 0,Y 317.776,Z 1111.989,A -85,B 0,C 180,E1 9956.59,E2 9956.59} C_VEL
LIN {X 0,Y 323.121,Z 1097.582,A -85,B 0,C 180,E1 9952.972,E2 9952.972} C_VEL
LIN {X 0,Y 328.748,Z 1082.895,A -85,B 0,C 180,E1 9949.851,E2 9949.851} C_VEL
LIN {X 0,Y 334.983,Z 1066.125,A -85,B 0,C 180,E1 9946.88,E2 9946.88} C_VEL
LIN {X 0,Y 341.675,Z 1047.7,A -85,B 0,C 180,E1 9944.144,E2 9944.144} C_VEL
LIN {X 0,Y 347.582,Z 1030.537,A -85,B 0,C 180,E1 9942.002,E2 9942.002} C_VEL
LIN {X 0,Y 353.931,Z 1010.513,A -85,B 0,C 180,E1 9939.915,E2 9939.915} C_VEL
LIN {X 0,Y 359.579,Z 991.128,A -85,B 0,C 180,E1 9938.23,E2 9938.23} C_VEL
LIN {X 0,Y 364.937,Z 969.94,A -85,B 0,C 180,E1 9936.736,E2 9936.736} C_VEL
LIN {X 0,Y 369.832,Z 947.595,A -85,B 0,C 180,E1 9935.467,E2 9935.467} C_VEL
LIN {X 0,Y 373.74,Z 925.795,A -85,B 0,C 180,E1 9934.505,E2 9934.505} C_VEL
LIN {X 0,Y 376.989,Z 902.23,A -85,B 0,C 180,E1 9933.741,E2 9933.741} C_VEL
LIN {X 0,Y 379.143,Z 878.169,A -85,B 0,C 180,E1 9933.17,E2 9933.17} C_VEL
LIN {X 0,Y 392.353,Z 669.491,A -85,B 0,C 180,E1 9928.933,E2 9928.933} C_VEL
LIN {X 0,Y 393.147,Z 656.081,A -85,B 0,C 180,E1 9928.646,E2 9928.646} C_VEL
LIN {X 0,Y 384.378,Z 642.214,A -85,B 0,C 180,E1 9925.871,E2 9925.871} C_VEL
LIN {X 0,Y 376.778,Z 630.99,A -85,B 0,C 180,E1 9923.166,E2 9923.166} C_VEL
LIN {X 0,Y 370.101,Z 621.755,A -85,B 0,C 180,E1 9920.478,E2 9920.478} C_VEL
LIN {X 0,Y 365.551,Z 615.777,A -85,B 0,C 180,E1 9918.416,E2 9918.416} C_VEL
LIN {X 0,Y 362.109,Z 611.407,A -85,B 0,C 180,E1 9916.688,E2 9916.688} C_VEL
LIN {X 0,Y 358.691,Z 607.089,A -85,B 0,C 180,E1 9914.777,E2 9914.777} C_VEL
LIN {X 0,Y 354.48,Z 601.941,A -85,B 0,C 180,E1 9912.047,E2 9912.047} C_VEL
LIN {X 0,Y 349.674,Z 596.323,A -85,B 0,C 180,E1 9908.054,E2 9908.054} C_VEL
LIN {X 0,Y 344.952,Z 591.653,A -85,B 0,C 180,E1 9901.162,E2 9901.162} C_VEL
LIN {X 0,Y 344.295,Z 591.034,A -85,B 0,C 180,E1 9897.836,E2 9897.836} C_VEL
LIN {X 0,Y 344.653,Z 592.378,A -85,B 0,C 180,E1 9894.172,E2 9894.172} C_VEL
LIN {X 0,Y 347.552,Z 596.016,A -85,B 0,C 180,E1 9888.817,E2 9888.817} C_VEL
LIN {X 0,Y 351.061,Z 600.847,A -85,B 0,C 180,E1 9885.147,E2 9885.147} C_VEL
LIN {X 0,Y 355.633,Z 607.294,A -85,B 0,C 180,E1 9881.646,E2 9881.646} C_VEL
LIN {X 0,Y 359.335,Z 612.409,A -85,B 0,C 180,E1 9879.348,E2 9879.348} C_VEL
LIN {X 0,Y 363.97,Z 618.966,A -85,B 0,C 180,E1 9876.869,E2 9876.869} C_VEL
LIN {X 0,Y 370.004,Z 627.84,A -85,B 0,C 180,E1 9874.081,E2 9874.081} C_VEL
LIN {X 0,Y 376.072,Z 637.139,A -85,B 0,C 180,E1 9871.629,E2 9871.629} C_VEL
LIN {X 0,Y 384.025,Z 649.92,A -85,B 0,C 180,E1 9868.793,E2 9868.793} C_VEL
LIN {X 0,Y 390.552,Z 661.394,A -85,B 0,C 180,E1 9866.691,E2 9866.691} C_VEL
LIN {X 0,Y 377.438,Z 891.676,A -85,B 0,C 180,E1 9862.276,E2 9862.276} C_VEL
LIN {X 0,Y 375.048,Z 914.688,A -85,B 0,C 180,E1 9861.686,E2 9861.686} C_VEL
LIN {X 0,Y 372.011,Z 934.774,A -85,B 0,C 180,E1 9860.964,E2 9860.964} C_VEL
LIN {X 0,Y 367.9,Z 955.884,A -85,B 0,C 180,E1 9859.95,E2 9859.95} C_VEL
LIN {X 0,Y 363.193,Z 976.008,A -85,B 0,C 180,E1 9858.726,E2 9858.726} C_VEL
LIN {X 0,Y 357.939,Z 994.958,A -85,B 0,C 180,E1 9857.279,E2 9857.279} C_VEL
LIN {X 0,Y 351.929,Z 1014.157,A -85,B 0,C 180,E1 9855.489,E2 9855.489} C_VEL
LIN {X 0,Y 345.635,Z 1032.464,A -85,B 0,C 180,E1 9853.408,E2 9853.408} C_VEL
LIN {X 0,Y 339.277,Z 1049.191,A -85,B 0,C 180,E1 9851.086,E2 9851.086} C_VEL
LIN {X 0,Y 332.523,Z 1065.98,A -85,B 0,C 180,E1 9848.274,E2 9848.274} C_VEL
LIN {X 0,Y 326.536,Z 1080.401,A -85,B 0,C 180,E1 9845.361,E2 9845.361} C_VEL
LIN {X 0,Y 321.007,Z 1093.329,A -85,B 0,C 180,E1 9842.183,E2 9842.183} C_VEL
LIN {X 0,Y 315.878,Z 1105.545,A -85,B 0,C 180,E1 9838.553,E2 9838.553} C_VEL
LIN {X 0,Y 311.794,Z 1115.828,A -85,B 0,C 180,E1 9834.834,E2 9834.834} C_VEL
LIN {X 0,Y 308.577,Z 1124.561,A -85,B 0,C 180,E1 9830.881,E2 9830.881} C_VEL
LIN {X 0,Y 306.277,Z 1131.865,A -85,B 0,C 180,E1 9826.695,E2 9826.695} C_VEL
LIN {X 0,Y 304.968,Z 1137.258,A -85,B 0,C 180,E1 9822.689,E2 9822.689} C_VEL
LIN {X 0,Y 304.3,Z 1140.996,A -85,B 0,C 180,E1 9818.693,E2 9818.693} C_VEL
LIN {X 0,Y 304.031,Z 1143.455,A -85,B 0,C 180,E1 9814.527,E2 9814.527} C_VEL
LIN {X 0,Y 303.983,Z 1144.309,A -85,B 0,C 180,E1 9810.942,E2 9810.942} C_VEL
LIN {X 0,Y 303.993,Z 1143.999,A -85,B 0,C 180,E1 9806.983,E2 9806.983} C_VEL
LIN {X 0,Y 304.142,Z 1142.318,A -85,B 0,C 180,E1 9803.131,E2 9803.131} C_VEL
LIN {X 0,Y 304.599,Z 1139.048,A -85,B 0,C 180,E1 9798.958,E2 9798.958} C_VEL
LIN {X 0,Y 305.602,Z 1134.507,A -85,B 0,C 180,E1 9795.021,E2 9795.021} C_VEL
LIN {X 0,Y 306.324,Z 1131.723,A -85,B 0,C 180,E1 9793.11,E2 9793.11} C_VEL
LIN {X 0,Y 306.004,Z 1129.652,A -85,B 0,C 180,E1 9791.712,E2 9791.712} C_VEL
LIN {X 0,Y 302.11,Z 1123.701,A -85,B 0,C 180,E1 9787.933,E2 9787.933} C_VEL
LIN {X 0,Y 302.287,Z 1121.431,A -85,B 0,C 180,E1 9786.743,E2 9786.743} C_VEL
LIN {X 0,Y 306.111,Z 1111.961,A -85,B 0,C 180,E1 9782.788,E2 9782.788} C_VEL
LIN {X 0,Y 311.164,Z 1100.333,A -85,B 0,C 180,E1 9778.846,E2 9778.846} C_VEL
LIN {X 0,Y 316.775,Z 1087.84,A -85,B 0,C 180,E1 9775.379,E2 9775.379} C_VEL
LIN {X 0,Y 322.622,Z 1074.615,A -85,B 0,C 180,E1 9772.372,E2 9772.372} C_VEL
LIN {X 0,Y 329.228,Z 1059.275,A -85,B 0,C 180,E1 9769.465,E2 9769.465} C_VEL
LIN {X 0,Y 335.933,Z 1043.045,A -85,B 0,C 180,E1 9766.915,E2 9766.915} C_VEL
LIN {X 0,Y 342.445,Z 1025.814,A -85,B 0,C 180,E1 9764.698,E2 9764.698} C_VEL
LIN {X 0,Y 349.062,Z 1006.756,A -85,B 0,C 180,E1 9762.676,E2 9762.676} C_VEL
LIN {X 0,Y 355.004,Z 987.625,A -85,B 0,C 180,E1 9761.014,E2 9761.014} C_VEL
LIN {X 0,Y 360.281,Z 967.757,A -85,B 0,C 180,E1 9759.635,E2 9759.635} C_VEL
LIN {X 0,Y 365.156,Z 945.977,A -85,B 0,C 180,E1 9758.431,E2 9758.431} C_VEL
LIN {X 0,Y 369.089,Z 924.258,A -85,B 0,C 180,E1 9757.52,E2 9757.52} C_VEL
LIN {X 0,Y 371.958,Z 902.197,A -85,B 0,C 180,E1 9756.865,E2 9756.865} C_VEL
LIN {X 0,Y 374.105,Z 872.834,A -85,B 0,C 180,E1 9756.242,E2 9756.242} C_VEL
LIN {X 0,Y 377.405,Z 814.059,A -85,B 0,C 180,E1 9755.104,E2 9755.104} C_VEL
LIN {X 0,Y 372.744,Z 831.422,A -85,B 0,C 180,E1 9754.565,E2 9754.565} C_VEL
LIN {X 0,Y 368.81,Z 842.602,A -85,B 0,C 180,E1 9753.974,E2 9753.974} C_VEL
LIN {X 0,Y 362.163,Z 871.561,A -85,B 0,C 180,E1 9753.285,E2 9753.285} C_VEL
LIN {X 0,Y 358.033,Z 885.746,A -85,B 0,C 180,E1 9752.71,E2 9752.71} C_VEL
LIN {X 0,Y 354.894,Z 894.118,A -85,B 0,C 180,E1 9752.221,E2 9752.221} C_VEL
LIN {X 0,Y 350.628,Z 909.159,A -85,B 0,C 180,E1 9751.889,E2 9751.889} C_VEL
LIN {X 0,Y 346.184,Z 919.933,A -85,B 0,C 180,E1 9751.422,E2 9751.422} C_VEL
LIN {X 0,Y 342.011,Z 927.297,A -85,B 0,C 180,E1 9750.82,E2 9750.82} C_VEL
LIN {X 0,Y 339.434,Z 931.103,A -85,B 0,C 180,E1 9750.405,E2 9750.405} C_VEL
LIN {X 0,Y 334.571,Z 940.162,A -85,B 0,C 180,E1 9749.841,E2 9749.841} C_VEL
LIN {X 0,Y 330.979,Z 945.344,A -85,B 0,C 180,E1 9749.301,E2 9749.301} C_VEL
LIN {X 0,Y 326.966,Z 949.785,A -85,B 0,C 180,E1 9748.493,E2 9748.493} C_VEL
LIN {X 0,Y 322.14,Z 956.634,A -85,B 0,C 180,E1 9747.799,E2 9747.799} C_VEL
LIN {X 0,Y 318.53,Z 960.557,A -85,B 0,C 180,E1 9747.075,E2 9747.075} C_VEL
LIN {X 0,Y 316.082,Z 962.583,A -85,B 0,C 180,E1 9746.464,E2 9746.464} C_VEL
LIN {X 0,Y 312.278,Z 967.259,A -85,B 0,C 180,E1 9745.814,E2 9745.814} C_VEL
LIN {X 0,Y 309.257,Z 969.964,A -85,B 0,C 180,E1 9745.058,E2 9745.058} C_VEL
LIN {X 0,Y 308.043,Z 971.055,A -85,B 0,C 180,E1 9744.549,E2 9744.549} C_VEL
LIN {X 0,Y 307.434,Z 975.083,A -85,B 0,C 180,E1 9743.988,E2 9743.988} C_VEL
LIN {X 0,Y 305.694,Z 990.23,A -85,B 0,C 180,E1 9741.994,E2 9741.994} C_VEL
LIN {X 0,Y 303.966,Z 1004.366,A -85,B 0,C 180,E1 9739.704,E2 9739.704} C_VEL
LIN {X 0,Y 302.454,Z 1016.36,A -85,B 0,C 180,E1 9737.309,E2 9737.309} C_VEL
LIN {X 0,Y 301.127,Z 1027.319,A -85,B 0,C 180,E1 9734.617,E2 9734.617} C_VEL
LIN {X 0,Y 300.147,Z 1036.218,A -85,B 0,C 180,E1 9731.92,E2 9731.92} C_VEL
LIN {X 0,Y 299.448,Z 1043.71,A -85,B 0,C 180,E1 9729.029,E2 9729.029} C_VEL
LIN {X 0,Y 299.073,Z 1049.751,A -85,B 0,C 180,E1 9725.949,E2 9725.949} C_VEL
LIN {X 0,Y 299.019,Z 1053.989,A -85,B 0,C 180,E1 9722.876,E2 9722.876} C_VEL
LIN {X 0,Y 299.227,Z 1056.467,A -85,B 0,C 180,E1 9719.809,E2 9719.809} C_VEL
LIN {X 0,Y 299.676,Z 1057.268,A -85,B 0,C 180,E1 9716.749,E2 9716.749} C_VEL
LIN {X 0,Y 300.428,Z 1056.397,A -85,B 0,C 180,E1 9713.695,E2 9713.695} C_VEL
LIN {X 0,Y 301.547,Z 1053.807,A -85,B 0,C 180,E1 9710.65,E2 9710.65} C_VEL
LIN {X 0,Y 303.106,Z 1049.148,A -85,B 0,C 180,E1 9707.534,E2 9707.534} C_VEL
LIN {X 0,Y 304.872,Z 1043.246,A -85,B 0,C 180,E1 9704.79,E2 9704.79} C_VEL
LIN {X 0,Y 306.918,Z 1035.783,A -85,B 0,C 180,E1 9702.169,E2 9702.169} C_VEL
LIN {X 0,Y 309.145,Z 1026.693,A -85,B 0,C 180,E1 9699.709,E2 9699.709} C_VEL
LIN {X 0,Y 311.594,Z 1015.767,A -85,B 0,C 180,E1 9697.353,E2 9697.353} C_VEL
LIN {X 0,Y 314.006,Z 1003.54,A -85,B 0,C 180,E1 9695.247,E2 9695.247} C_VEL
LIN {X 0,Y 316.455,Z 988.909,A -85,B 0,C 180,E1 9693.242,E2 9693.242} C_VEL
LIN {X 0,Y 317.087,Z 986.57,A -85,B 0,C 180,E1 9692.894,E2 9692.894} C_VEL
LIN {X 0,Y 320.719,Z 983.851,A -85,B 0,C 180,E1 9692.12,E2 9692.12} C_VEL
LIN {X 0,Y 324.608,Z 980.125,A -85,B 0,C 180,E1 9691.583,E2 9691.583} C_VEL
LIN {X 0,Y 328.79,Z 976.98,A -85,B 0,C 180,E1 9690.886,E2 9690.886} C_VEL
LIN {X 0,Y 333.339,Z 972.019,A -85,B 0,C 180,E1 9690.336,E2 9690.336} C_VEL
LIN {X 0,Y 337.315,Z 968.535,A -85,B 0,C 180,E1 9689.742,E2 9689.742} C_VEL
LIN {X 0,Y 342.207,Z 962.976,A -85,B 0,C 180,E1 9689.206,E2 9689.206} C_VEL
LIN {X 0,Y 344,Z 960.591,A -85,B 0,C 180,E1 9689.03,E2 9689.03} C_VEL
LIN {X 0,Y 349.18,Z 954.909,A -85,B 0,C 180,E1 9688.399,E2 9688.399} C_VEL
LIN {X 0,Y 354.249,Z 947.683,A -85,B 0,C 180,E1 9687.953,E2 9687.953} C_VEL
LIN {X 0,Y 356.853,Z 943.542,A -85,B 0,C 180,E1 9687.741,E2 9687.741} C_VEL
LIN {X 0,Y 362.322,Z 935.729,A -85,B 0,C 180,E1 9687.21,E2 9687.21} C_VEL
LIN {X 0,Y 367.629,Z 925.374,A -85,B 0,C 180,E1 9686.849,E2 9686.849} C_VEL
LIN {X 0,Y 370.027,Z 919.792,A -85,B 0,C 180,E1 9686.722,E2 9686.722} C_VEL
LIN {X 0,Y 366.006,Z 942.669,A -85,B 0,C 180,E1 9685.779,E2 9685.779} C_VEL
LIN {X 0,Y 361.546,Z 963.63,A -85,B 0,C 180,E1 9684.669,E2 9684.669} C_VEL
LIN {X 0,Y 356.222,Z 984.395,A -85,B 0,C 180,E1 9683.284,E2 9683.284} C_VEL
LIN {X 0,Y 350.195,Z 1005.323,A -85,B 0,C 180,E1 9681.576,E2 9681.576} C_VEL
LIN {X 0,Y 344.055,Z 1024.309,A -85,B 0,C 180,E1 9679.686,E2 9679.686} C_VEL
LIN {X 0,Y 337.197,Z 1043.877,A -85,B 0,C 180,E1 9677.339,E2 9677.339} C_VEL
LIN {X 0,Y 330.613,Z 1061.577,A -85,B 0,C 180,E1 9674.802,E2 9674.802} C_VEL
LIN {X 0,Y 324.15,Z 1077.943,A -85,B 0,C 180,E1 9671.981,E2 9671.981} C_VEL
LIN {X 0,Y 317.826,Z 1093.886,A -85,B 0,C 180,E1 9668.723,E2 9668.723} C_VEL
LIN {X 0,Y 312.405,Z 1107.494,A -85,B 0,C 180,E1 9665.401,E2 9665.401} C_VEL
LIN {X 0,Y 307.3,Z 1120.802,A -85,B 0,C 180,E1 9661.52,E2 9661.52} C_VEL
LIN {X 0,Y 303.223,Z 1132.347,A -85,B 0,C 180,E1 9657.493,E2 9657.493} C_VEL
LIN {X 0,Y 300.148,Z 1141.982,A -85,B 0,C 180,E1 9653.354,E2 9653.354} C_VEL
LIN {X 0,Y 297.967,Z 1150.281,A -85,B 0,C 180,E1 9648.996,E2 9648.996} C_VEL
LIN {X 0,Y 296.78,Z 1156.207,A -85,B 0,C 180,E1 9645.035,E2 9645.035} C_VEL
LIN {X 0,Y 296.147,Z 1161.132,A -85,B 0,C 180,E1 9640.702,E2 9640.702} C_VEL
LIN {X 0,Y 295.965,Z 1163.994,A -85,B 0,C 180,E1 9636.986,E2 9636.986} C_VEL
LIN {X 0,Y 295.944,Z 1165.71,A -85,B 0,C 180,E1 9633.293,E2 9633.293} C_VEL
LIN {X 0,Y 295.956,Z 1166.169,A -85,B 0,C 180,E1 9629.419,E2 9629.419} C_VEL
LIN {X 0,Y 295.959,Z 1165.419,A -85,B 0,C 180,E1 9625.932,E2 9625.932} C_VEL
LIN {X 0,Y 295.988,Z 1163.505,A -85,B 0,C 180,E1 9622.234,E2 9622.234} C_VEL
LIN {X 0,Y 296.294,Z 1159.731,A -85,B 0,C 180,E1 9617.923,E2 9617.923} C_VEL
LIN {X 0,Y 296.968,Z 1155.124,A -85,B 0,C 180,E1 9614.174,E2 9614.174} C_VEL
LIN {X 0,Y 298.53,Z 1147.945,A -85,B 0,C 180,E1 9609.683,E2 9609.683} C_VEL
LIN {X 0,Y 300.825,Z 1139.722,A -85,B 0,C 180,E1 9605.601,E2 9605.601} C_VEL
LIN {X 0,Y 304.099,Z 1129.657,A -85,B 0,C 180,E1 9601.526,E2 9601.526} C_VEL
LIN {X 0,Y 308.301,Z 1118.2,A -85,B 0,C 180,E1 9597.648,E2 9597.648} C_VEL
LIN {X 0,Y 313.259,Z 1105.279,A -85,B 0,C 180,E1 9594.035,E2 9594.035} C_VEL
LIN {X 0,Y 319.197,Z 1090.368,A -85,B 0,C 180,E1 9590.514,E2 9590.514} C_VEL
LIN {X 0,Y 325.126,Z 1075.447,A -85,B 0,C 180,E1 9587.566,E2 9587.566} C_VEL
LIN {X 0,Y 331.857,Z 1058.082,A -85,B 0,C 180,E1 9584.679,E2 9584.679} C_VEL
LIN {X 0,Y 338.575,Z 1040.042,A -85,B 0,C 180,E1 9582.163,E2 9582.163} C_VEL
LIN {X 0,Y 345.097,Z 1021.011,A -85,B 0,C 180,E1 9579.973,E2 9579.973} C_VEL
LIN {X 0,Y 351.563,Z 1000.607,A -85,B 0,C 180,E1 9578.019,E2 9578.019} C_VEL
LIN {X 0,Y 357.001,Z 981.353,A -85,B 0,C 180,E1 9576.505,E2 9576.505} C_VEL
LIN {X 0,Y 362.391,Z 959.514,A -85,B 0,C 180,E1 9575.108,E2 9575.108} C_VEL
LIN {X 0,Y 366.636,Z 939.225,A -85,B 0,C 180,E1 9574.069,E2 9574.069} C_VEL
LIN {X 0,Y 370.384,Z 916.881,A -85,B 0,C 180,E1 9573.191,E2 9573.191} C_VEL
LIN {X 0,Y 373.307,Z 893.862,A -85,B 0,C 180,E1 9572.521,E2 9572.521} C_VEL
LIN {X 0,Y 378.509,Z 816.508,A -85,B 0,C 180,E1 9570.905,E2 9570.905} C_VEL
LIN {X 0,Y 388.819,Z 660.483,A -85,B 0,C 180,E1 9567.739,E2 9567.739} C_VEL
LIN {X 0,Y 380.227,Z 646.77,A -85,B 0,C 180,E1 9564.881,E2 9564.881} C_VEL
LIN {X 0,Y 371.939,Z 634.399,A -85,B 0,C 180,E1 9561.734,E2 9561.734} C_VEL
LIN {X 0,Y 364.695,Z 624.471,A -85,B 0,C 180,E1 9558.543,E2 9558.543} C_VEL
LIN {X 0,Y 360.389,Z 618.934,A -85,B 0,C 180,E1 9556.355,E2 9556.355} C_VEL
LIN {X 0,Y 356.915,Z 614.492,A -85,B 0,C 180,E1 9554.354,E2 9554.354} C_VEL
LIN {X 0,Y 353.045,Z 609.632,A -85,B 0,C 180,E1 9551.765,E2 9551.765} C_VEL
LIN {X 0,Y 348.363,Z 604.062,A -85,B 0,C 180,E1 9547.752,E2 9547.752} C_VEL
LIN {X 0,Y 343.92,Z 599.539,A -85,B 0,C 180,E1 9540.999,E2 9540.999} C_VEL
LIN {X 0,Y 343.312,Z 598.998,A -85,B 0,C 180,E1 9537.663,E2 9537.663} C_VEL
LIN {X 0,Y 343.726,Z 600.467,A -85,B 0,C 180,E1 9533.989,E2 9533.989} C_VEL
LIN {X 0,Y 346.403,Z 603.864,A -85,B 0,C 180,E1 9529.017,E2 9529.017} C_VEL
LIN {X 0,Y 349.922,Z 608.741,A -85,B 0,C 180,E1 9525.267,E2 9525.267} C_VEL
LIN {X 0,Y 354.199,Z 615.047,A -85,B 0,C 180,E1 9521.909,E2 9521.909} C_VEL
LIN {X 0,Y 357.705,Z 620.003,A -85,B 0,C 180,E1 9519.677,E2 9519.677} C_VEL
LIN {X 0,Y 362.24,Z 626.546,A -85,B 0,C 180,E1 9517.19,E2 9517.19} C_VEL
LIN {X 0,Y 368.107,Z 635.383,A -85,B 0,C 180,E1 9514.413,E2 9514.413} C_VEL
LIN {X 0,Y 374.93,Z 646.029,A -85,B 0,C 180,E1 9511.617,E2 9511.617} C_VEL
LIN {X 0,Y 382.827,Z 659.328,A -85,B 0,C 180,E1 9508.772,E2 9508.772} C_VEL
LIN {X 0,Y 386.248,Z 665.615,A -85,B 0,C 180,E1 9507.633,E2 9507.633} C_VEL
LIN {X 0,Y 372.752,Z 892.901,A -85,B 0,C 180,E1 9503.254,E2 9503.254} C_VEL
LIN {X 0,Y 370.133,Z 916.385,A -85,B 0,C 180,E1 9502.636,E2 9502.636} C_VEL
LIN {X 0,Y 366.926,Z 936.709,A -85,B 0,C 180,E1 9501.891,E2 9501.891} C_VEL
LIN {X 0,Y 362.707,Z 957.212,A -85,B 0,C 180,E1 9500.884,E2 9500.884} C_VEL
LIN {X 0,Y 357.689,Z 977.63,A -85,B 0,C 180,E1 9499.617,E2 9499.617} C_VEL
LIN {X 0,Y 352.308,Z 996.338,A -85,B 0,C 180,E1 9498.169,E2 9498.169} C_VEL
LIN {X 0,Y 346.054,Z 1015.434,A -85,B 0,C 180,E1 9496.355,E2 9496.355} C_VEL
LIN {X 0,Y 339.862,Z 1032.75,A -85,B 0,C 180,E1 9494.365,E2 9494.365} C_VEL
LIN {X 0,Y 333.203,Z 1049.601,A -85,B 0,C 180,E1 9492.003,E2 9492.003} C_VEL
LIN {X 0,Y 326.17,Z 1066.354,A -85,B 0,C 180,E1 9489.16,E2 9489.16} C_VEL
LIN {X 0,Y 319.907,Z 1080.75,A -85,B 0,C 180,E1 9486.208,E2 9486.208} C_VEL
LIN {X 0,Y 314.112,Z 1093.672,A -85,B 0,C 180,E1 9482.978,E2 9482.978} C_VEL
LIN {X 0,Y 308.706,Z 1105.873,A -85,B 0,C 180,E1 9479.28,E2 9479.28} C_VEL
LIN {X 0,Y 304.384,Z 1116.13,A -85,B 0,C 180,E1 9475.488,E2 9475.488} C_VEL
LIN {X 0,Y 300.95,Z 1124.875,A -85,B 0,C 180,E1 9471.436,E2 9471.436} C_VEL
LIN {X 0,Y 298.485,Z 1132.171,A -85,B 0,C 180,E1 9467.144,E2 9467.144} C_VEL
LIN {X 0,Y 297.061,Z 1137.557,A -85,B 0,C 180,E1 9463.033,E2 9463.033} C_VEL
LIN {X 0,Y 296.336,Z 1141.292,A -85,B 0,C 180,E1 9458.929,E2 9458.929} C_VEL
LIN {X 0,Y 296.04,Z 1143.747,A -85,B 0,C 180,E1 9454.649,E2 9454.649} C_VEL
LIN {X 0,Y 295.989,Z 1144.6,A -85,B 0,C 180,E1 9450.968,E2 9450.968} C_VEL
LIN {X 0,Y 296.001,Z 1144.291,A -85,B 0,C 180,E1 9446.902,E2 9446.902} C_VEL
LIN {X 0,Y 296.158,Z 1142.649,A -85,B 0,C 180,E1 9443.016,E2 9443.016} C_VEL
LIN {X 0,Y 296.656,Z 1139.413,A -85,B 0,C 180,E1 9438.727,E2 9438.727} C_VEL
LIN {X 0,Y 297.755,Z 1134.807,A -85,B 0,C 180,E1 9434.616,E2 9434.616} C_VEL
LIN {X 0,Y 299.649,Z 1128.581,A -85,B 0,C 180,E1 9430.508,E2 9430.508} C_VEL
LIN {X 0,Y 302.287,Z 1121.431,A -85,B 0,C 180,E1 9426.743,E2 9426.743} C_VEL
LIN {X 0,Y 302.493,Z 1118.69,A -85,B 0,C 180,E1 9425.366,E2 9425.366} C_VEL
LIN {X 0,Y 300.134,Z 1110.992,A -85,B 0,C 180,E1 9421.625,E2 9421.625} C_VEL
LIN {X 0,Y 300.771,Z 1108.032,A -85,B 0,C 180,E1 9420.492,E2 9420.492} C_VEL
LIN {X 0,Y 306.245,Z 1096.359,A -85,B 0,C 180,E1 9416.735,E2 9416.735} C_VEL
LIN {X 0,Y 312.143,Z 1083.697,A -85,B 0,C 180,E1 9413.43,E2 9413.43} C_VEL
LIN {X 0,Y 319.23,Z 1068.304,A -85,B 0,C 180,E1 9410.118,E2 9410.118} C_VEL
LIN {X 0,Y 326.178,Z 1052.679,A -85,B 0,C 180,E1 9407.355,E2 9407.355} C_VEL
LIN {X 0,Y 332.903,Z 1036.323,A -85,B 0,C 180,E1 9404.983,E2 9404.983} C_VEL
LIN {X 0,Y 339.884,Z 1017.956,A -85,B 0,C 180,E1 9402.779,E2 9402.779} C_VEL
LIN {X 0,Y 346.364,Z 999.244,A -85,B 0,C 180,E1 9400.942,E2 9400.942} C_VEL
LIN {X 0,Y 352.092,Z 980.13,A -85,B 0,C 180,E1 9399.428,E2 9399.428} C_VEL
LIN {X 0,Y 357.581,Z 959.004,A -85,B 0,C 180,E1 9398.082,E2 9398.082} C_VEL
LIN {X 0,Y 361.734,Z 939.737,A -85,B 0,C 180,E1 9397.114,E2 9397.114} C_VEL
LIN {X 0,Y 365.385,Z 918.221,A -85,B 0,C 180,E1 9396.295,E2 9396.295} C_VEL
LIN {X 0,Y 368.099,Z 896.273,A -85,B 0,C 180,E1 9395.691,E2 9395.691} C_VEL
LIN {X 0,Y 370.809,Z 853.128,A -85,B 0,C 180,E1 9394.824,E2 9394.824} C_VEL
LIN {X 0,Y 365.641,Z 875.018,A -85,B 0,C 180,E1 9394.298,E2 9394.298} C_VEL
LIN {X 0,Y 361.335,Z 889.182,A -85,B 0,C 180,E1 9393.734,E2 9393.734} C_VEL
LIN {X 0,Y 358.36,Z 897.075,A -85,B 0,C 180,E1 9393.295,E2 9393.295} C_VEL
LIN {X 0,Y 353.976,Z 911.753,A -85,B 0,C 180,E1 9392.992,E2 9392.992} C_VEL
LIN {X 0,Y 349.089,Z 923.311,A -85,B 0,C 180,E1 9392.519,E2 9392.519} C_VEL
LIN {X 0,Y 344.298,Z 931.466,A -85,B 0,C 180,E1 9391.907,E2 9391.907} C_VEL
LIN {X 0,Y 341.423,Z 935.809,A -85,B 0,C 180,E1 9391.48,E2 9391.48} C_VEL
LIN {X 0,Y 335.962,Z 945.189,A -85,B 0,C 180,E1 9390.89,E2 9390.89} C_VEL
LIN {X 0,Y 331.546,Z 951.226,A -85,B 0,C 180,E1 9390.241,E2 9390.241} C_VEL
LIN {X 0,Y 327.476,Z 955.533,A -85,B 0,C 180,E1 9389.521,E2 9389.521} C_VEL
LIN {X 0,Y 322.923,Z 961.745,A -85,B 0,C 180,E1 9388.883,E2 9388.883} C_VEL
LIN {X 0,Y 318.364,Z 966.453,A -85,B 0,C 180,E1 9388.052,E2 9388.052} C_VEL
LIN {X 0,Y 316.01,Z 968.321,A -85,B 0,C 180,E1 9387.513,E2 9387.513} C_VEL
LIN {X 0,Y 311.39,Z 973.608,A -85,B 0,C 180,E1 9386.714,E2 9386.714} C_VEL
LIN {X 0,Y 307.678,Z 976.669,A -85,B 0,C 180,E1 9385.815,E2 9385.815} C_VEL
LIN {X 0,Y 306.623,Z 977.247,A -85,B 0,C 180,E1 9385.496,E2 9385.496} C_VEL
LIN {X 0,Y 302.719,Z 981.298,A -85,B 0,C 180,E1 9384.727,E2 9384.727} C_VEL
LIN {X 0,Y 300.107,Z 983.226,A -85,B 0,C 180,E1 9383.983,E2 9383.983} C_VEL
LIN {X 0,Y 298.997,Z 984.191,A -85,B 0,C 180,E1 9383.45,E2 9383.45} C_VEL
LIN {X 0,Y 296.488,Z 1003.093,A -85,B 0,C 180,E1 9380.429,E2 9380.429} C_VEL
LIN {X 0,Y 294.877,Z 1015.66,A -85,B 0,C 180,E1 9377.973,E2 9377.973} C_VEL
LIN {X 0,Y 293.541,Z 1026.366,A -85,B 0,C 180,E1 9375.408,E2 9375.408} C_VEL
LIN {X 0,Y 292.384,Z 1036.314,A -85,B 0,C 180,E1 9372.442,E2 9372.442} C_VEL
LIN {X 0,Y 291.624,Z 1044.181,A -85,B 0,C 180,E1 9369.473,E2 9369.473} C_VEL
LIN {X 0,Y 291.2,Z 1050.515,A -85,B 0,C 180,E1 9366.309,E2 9366.309} C_VEL
LIN {X 0,Y 291.12,Z 1055.009,A -85,B 0,C 180,E1 9363.151,E2 9363.151} C_VEL
LIN {X 0,Y 291.336,Z 1057.807,A -85,B 0,C 180,E1 9360.001,E2 9360.001} C_VEL
LIN {X 0,Y 291.813,Z 1058.876,A -85,B 0,C 180,E1 9356.858,E2 9356.858} C_VEL
LIN {X 0,Y 292.604,Z 1058.237,A -85,B 0,C 180,E1 9353.723,E2 9353.723} C_VEL
LIN {X 0,Y 293.789,Z 1055.902,A -85,B 0,C 180,E1 9350.599,E2 9350.599} C_VEL
LIN {X 0,Y 295.296,Z 1052.056,A -85,B 0,C 180,E1 9347.684,E2 9347.684} C_VEL
LIN {X 0,Y 297.191,Z 1046.4,A -85,B 0,C 180,E1 9344.787,E2 9344.787} C_VEL
LIN {X 0,Y 299.488,Z 1038.764,A -85,B 0,C 180,E1 9341.912,E2 9341.912} C_VEL
LIN {X 0,Y 301.841,Z 1030.318,A -85,B 0,C 180,E1 9339.444,E2 9339.444} C_VEL
LIN {X 0,Y 304.693,Z 1018.73,A -85,B 0,C 180,E1 9336.811,E2 9336.811} C_VEL
LIN {X 0,Y 307.402,Z 1006.3,A -85,B 0,C 180,E1 9334.575,E2 9334.575} C_VEL
LIN {X 0,Y 309.293,Z 997.605,A -85,B 0,C 180,E1 9333.221,E2 9333.221} C_VEL
LIN {X 0,Y 312.966,Z 995.222,A -85,B 0,C 180,E1 9332.404,E2 9332.404} C_VEL
LIN {X 0,Y 316.298,Z 992.466,A -85,B 0,C 180,E1 9331.901,E2 9331.901} C_VEL
LIN {X 0,Y 320.763,Z 989.506,A -85,B 0,C 180,E1 9331.109,E2 9331.109} C_VEL
LIN {X 0,Y 325.136,Z 985.63,A -85,B 0,C 180,E1 9330.492,E2 9330.492} C_VEL
LIN {X 0,Y 329.848,Z 981.87,A -85,B 0,C 180,E1 9329.789,E2 9329.789} C_VEL
LIN {X 0,Y 334.527,Z 977.226,A -85,B 0,C 180,E1 9329.264,E2 9329.264} C_VEL
LIN {X 0,Y 339.857,Z 972.294,A -85,B 0,C 180,E1 9328.56,E2 9328.56} C_VEL
LIN {X 0,Y 346.4,Z 964.855,A -85,B 0,C 180,E1 9327.921,E2 9327.921} C_VEL
LIN {X 0,Y 351.854,Z 958.734,A -85,B 0,C 180,E1 9327.322,E2 9327.322} C_VEL
LIN {X 0,Y 357.708,Z 950.509,A -85,B 0,C 180,E1 9326.876,E2 9326.876} C_VEL
LIN {X 0,Y 359.731,Z 947.484,A -85,B 0,C 180,E1 9326.706,E2 9326.706} C_VEL
LIN {X 0,Y 360.499,Z 946.493,A -85,B 0,C 180,E1 9326.627,E2 9326.627} C_VEL
LIN {X 0,Y 355.241,Z 969.221,A -85,B 0,C 180,E1 9325.352,E2 9325.352} C_VEL
LIN {X 0,Y 349.522,Z 990.415,A -85,B 0,C 180,E1 9323.865,E2 9323.865} C_VEL
LIN {X 0,Y 343.283,Z 1010.401,A -85,B 0,C 180,E1 9322.123,E2 9322.123} C_VEL
LIN {X 0,Y 336.524,Z 1030.161,A -85,B 0,C 180,E1 9320.046,E2 9320.046} C_VEL
LIN {X 0,Y 330.018,Z 1047.619,A -85,B 0,C 180,E1 9317.833,E2 9317.833} C_VEL
LIN {X 0,Y 322.786,Z 1065.848,A -85,B 0,C 180,E1 9315.07,E2 9315.07} C_VEL
LIN {X 0,Y 316.095,Z 1082.177,A -85,B 0,C 180,E1 9312.113,E2 9312.113} C_VEL
LIN {X 0,Y 309.672,Z 1097.381,A -85,B 0,C 180,E1 9308.784,E2 9308.784} C_VEL
LIN {X 0,Y 303.597,Z 1111.981,A -85,B 0,C 180,E1 9304.963,E2 9304.963} C_VEL
LIN {X 0,Y 298.861,Z 1123.849,A -85,B 0,C 180,E1 9301.236,E2 9301.236} C_VEL
LIN {X 0,Y 294.757,Z 1134.902,A -85,B 0,C 180,E1 9297.036,E2 9297.036} C_VEL
LIN {X 0,Y 291.766,Z 1144.18,A -85,B 0,C 180,E1 9292.783,E2 9292.783} C_VEL
LIN {X 0,Y 289.769,Z 1151.567,A -85,B 0,C 180,E1 9288.509,E2 9288.509} C_VEL
LIN {X 0,Y 288.616,Z 1157.465,A -85,B 0,C 180,E1 9284.239,E2 9284.239} C_VEL
LIN {X 0,Y 288.1,Z 1161.513,A -85,B 0,C 180,E1 9280.195,E2 9280.195} C_VEL
LIN {X 0,Y 287.976,Z 1164.063,A -85,B 0,C 180,E1 9276.579,E2 9276.579} C_VEL
LIN {X 0,Y 287.967,Z 1165.661,A -85,B 0,C 180,E1 9272.388,E2 9272.388} C_VEL
LIN {X 0,Y 287.969,Z 1165.807,A -85,B 0,C 180,E1 9268.806,E2 9268.806} C_VEL
LIN {X 0,Y 287.962,Z 1164.905,A -85,B 0,C 180,E1 9265.21,E2 9265.21} C_VEL
LIN {X 0,Y 288.051,Z 1162.525,A -85,B 0,C 180,E1 9261.014,E2 9261.014} C_VEL
LIN {X 0,Y 288.42,Z 1158.729,A -85,B 0,C 180,E1 9256.937,E2 9256.937} C_VEL
LIN {X 0,Y 289.44,Z 1153.15,A -85,B 0,C 180,E1 9252.51,E2 9252.51} C_VEL
LIN {X 0,Y 291.203,Z 1146.019,A -85,B 0,C 180,E1 9248.234,E2 9248.234} C_VEL
LIN {X 0,Y 294.095,Z 1136.799,A -85,B 0,C 180,E1 9243.77,E2 9243.77} C_VEL
LIN {X 0,Y 297.565,Z 1127.174,A -85,B 0,C 180,E1 9239.956,E2 9239.956} C_VEL
LIN {X 0,Y 302.518,Z 1114.583,A -85,B 0,C 180,E1 9235.815,E2 9235.815} C_VEL
LIN {X 0,Y 308.042,Z 1101.292,A -85,B 0,C 180,E1 9232.159,E2 9232.159} C_VEL
LIN {X 0,Y 314.213,Z 1086.501,A -85,B 0,C 180,E1 9228.799,E2 9228.799} C_VEL
LIN {X 0,Y 321.156,Z 1069.773,A -85,B 0,C 180,E1 9225.605,E2 9225.605} C_VEL
LIN {X 0,Y 327.839,Z 1053.1,A -85,B 0,C 180,E1 9222.949,E2 9222.949} C_VEL
LIN {X 0,Y 334.708,Z 1034.964,A -85,B 0,C 180,E1 9220.541,E2 9220.541} C_VEL
LIN {X 0,Y 341.429,Z 1016.013,A -85,B 0,C 180,E1 9218.43,E2 9218.43} C_VEL
LIN {X 0,Y 347.649,Z 996.362,A -85,B 0,C 180,E1 9216.638,E2 9216.638} C_VEL
LIN {X 0,Y 353.622,Z 975.382,A -85,B 0,C 180,E1 9215.059,E2 9215.059} C_VEL
LIN {X 0,Y 358.631,Z 954.823,A -85,B 0,C 180,E1 9213.817,E2 9213.817} C_VEL
LIN {X 0,Y 363.394,Z 931.265,A -85,B 0,C 180,E1 9212.699,E2 9212.699} C_VEL
LIN {X 0,Y 366.931,Z 909.392,A -85,B 0,C 180,E1 9211.92,E2 9211.92} C_VEL
LIN {X 0,Y 369.449,Z 886.005,A -85,B 0,C 180,E1 9211.319,E2 9211.319} C_VEL
LIN {X 0,Y 383.26,Z 683.331,A -85,B 0,C 180,E1 9207.17,E2 9207.17} C_VEL
LIN {X 0,Y 384.44,Z 664.7,A -85,B 0,C 180,E1 9206.764,E2 9206.764} C_VEL
LIN {X 0,Y 376.829,Z 652.435,A -85,B 0,C 180,E1 9204.111,E2 9204.111} C_VEL
LIN {X 0,Y 369.5,Z 641.294,A -85,B 0,C 180,E1 9201.218,E2 9201.218} C_VEL
LIN {X 0,Y 362.599,Z 631.62,A -85,B 0,C 180,E1 9198.072,E2 9198.072} C_VEL
LIN {X 0,Y 358.268,Z 625.936,A -85,B 0,C 180,E1 9195.789,E2 9195.789} C_VEL
LIN {X 0,Y 355.283,Z 622.029,A -85,B 0,C 180,E1 9194.006,E2 9194.006} C_VEL
LIN {X 0,Y 351.618,Z 617.322,A -85,B 0,C 180,E1 9191.481,E2 9191.481} C_VEL
LIN {X 0,Y 347.222,Z 611.934,A -85,B 0,C 180,E1 9187.611,E2 9187.611} C_VEL
LIN {X 0,Y 342.89,Z 607.425,A -85,B 0,C 180,E1 9180.835,E2 9180.835} C_VEL
LIN {X 0,Y 342.337,Z 606.942,A -85,B 0,C 180,E1 9177.656,E2 9177.656} C_VEL
LIN {X 0,Y 342.756,Z 608.452,A -85,B 0,C 180,E1 9173.971,E2 9173.971} C_VEL
LIN {X 0,Y 345.305,Z 611.813,A -85,B 0,C 180,E1 9169.151,E2 9169.151} C_VEL
LIN {X 0,Y 349.03,Z 617.197,A -85,B 0,C 180,E1 9165.144,E2 9165.144} C_VEL
LIN {X 0,Y 352.773,Z 622.793,A -85,B 0,C 180,E1 9162.175,E2 9162.175} C_VEL
LIN {X 0,Y 356.027,Z 627.489,A -85,B 0,C 180,E1 9160.049,E2 9160.049} C_VEL
LIN {X 0,Y 360.553,Z 634.163,A -85,B 0,C 180,E1 9157.499,E2 9157.499} C_VEL
LIN {X 0,Y 366.893,Z 643.894,A -85,B 0,C 180,E1 9154.452,E2 9154.452} C_VEL
LIN {X 0,Y 374.313,Z 656.071,A -85,B 0,C 180,E1 9151.392,E2 9151.392} C_VEL
LIN {X 0,Y 381.72,Z 669.012,A -85,B 0,C 180,E1 9148.715,E2 9148.715} C_VEL
LIN {X 0,Y 382.033,Z 670.02,A -85,B 0,C 180,E1 9148.592,E2 9148.592} C_VEL
LIN {X 0,Y 368.205,Z 893.736,A -85,B 0,C 180,E1 9144.265,E2 9144.265} C_VEL
LIN {X 0,Y 365.534,Z 916.633,A -85,B 0,C 180,E1 9143.656,E2 9143.656} C_VEL
LIN {X 0,Y 362.079,Z 937.689,A -85,B 0,C 180,E1 9142.88,E2 9142.88} C_VEL
LIN {X 0,Y 357.735,Z 957.995,A -85,B 0,C 180,E1 9141.873,E2 9141.873} C_VEL
LIN {X 0,Y 352.149,Z 979.673,A -85,B 0,C 180,E1 9140.505,E2 9140.505} C_VEL
LIN {X 0,Y 346.448,Z 998.756,A -85,B 0,C 180,E1 9138.999,E2 9138.999} C_VEL
LIN {X 0,Y 340.054,Z 1017.289,A -85,B 0,C 180,E1 9137.19,E2 9137.19} C_VEL
LIN {X 0,Y 333.111,Z 1035.663,A -85,B 0,C 180,E1 9135.003,E2 9135.003} C_VEL
LIN {X 0,Y 326.329,Z 1052.177,A -85,B 0,C 180,E1 9132.62,E2 9132.62} C_VEL
LIN {X 0,Y 319.49,Z 1067.628,A -85,B 0,C 180,E1 9129.908,E2 9129.908} C_VEL
LIN {X 0,Y 312.988,Z 1081.846,A -85,B 0,C 180,E1 9126.911,E2 9126.911} C_VEL
LIN {X 0,Y 306.97,Z 1094.692,A -85,B 0,C 180,E1 9123.623,E2 9123.623} C_VEL
LIN {X 0,Y 301.582,Z 1106.199,A -85,B 0,C 180,E1 9120.041,E2 9120.041} C_VEL
LIN {X 0,Y 297.009,Z 1116.445,A -85,B 0,C 180,E1 9116.168,E2 9116.168} C_VEL
LIN {X 0,Y 293.347,Z 1125.202,A -85,B 0,C 180,E1 9112.012,E2 9112.012} C_VEL
LIN {X 0,Y 290.71,Z 1132.475,A -85,B 0,C 180,E1 9107.618,E2 9107.618} C_VEL
LIN {X 0,Y 289.165,Z 1137.855,A -85,B 0,C 180,E1 9103.395,E2 9103.395} C_VEL
LIN {X 0,Y 288.373,Z 1141.588,A -85,B 0,C 180,E1 9099.177,E2 9099.177} C_VEL
LIN {X 0,Y 288.049,Z 1144.039,A -85,B 0,C 180,E1 9094.779,E2 9094.779} C_VEL
LIN {X 0,Y 287.994,Z 1144.891,A -85,B 0,C 180,E1 9090.995,E2 9090.995} C_VEL
LIN {X 0,Y 288.009,Z 1144.582,A -85,B 0,C 180,E1 9086.816,E2 9086.816} C_VEL
LIN {X 0,Y 288.177,Z 1142.944,A -85,B 0,C 180,E1 9082.825,E2 9082.825} C_VEL
LIN {X 0,Y 288.731,Z 1139.71,A -85,B 0,C 180,E1 9078.413,E2 9078.413} C_VEL
LIN {X 0,Y 289.919,Z 1135.106,A -85,B 0,C 180,E1 9074.19,E2 9074.19} C_VEL
LIN {X 0,Y 291.958,Z 1128.887,A -85,B 0,C 180,E1 9069.973,E2 9069.973} C_VEL
LIN {X 0,Y 295.056,Z 1121.061,A -85,B 0,C 180,E1 9065.793,E2 9065.793} C_VEL
LIN {X 0,Y 299.3,Z 1111.287,A -85,B 0,C 180,E1 9061.681,E2 9061.681} C_VEL
LIN {X 0,Y 300.771,Z 1108.032,A -85,B 0,C 180,E1 9060.492,E2 9060.492} C_VEL
LIN {X 0,Y 301.513,Z 1104.588,A -85,B 0,C 180,E1 9059.182,E2 9059.182} C_VEL
LIN {X 0,Y 300.735,Z 1095.259,A -85,B 0,C 180,E1 9055.554,E2 9055.554} C_VEL
LIN {X 0,Y 301.831,Z 1091.731,A -85,B 0,C 180,E1 9054.492,E2 9054.492} C_VEL
LIN {X 0,Y 308.845,Z 1077.418,A -85,B 0,C 180,E1 9050.985,E2 9050.985} C_VEL
LIN {X 0,Y 315.947,Z 1062.508,A -85,B 0,C 180,E1 9047.985,E2 9047.985} C_VEL
LIN {X 0,Y 323.065,Z 1046.559,A -85,B 0,C 180,E1 9045.368,E2 9045.368} C_VEL
LIN {X 0,Y 330.535,Z 1028.595,A -85,B 0,C 180,E1 9042.942,E2 9042.942} C_VEL
LIN {X 0,Y 337.195,Z 1011.189,A -85,B 0,C 180,E1 9041.005,E2 9041.005} C_VEL
LIN {X 0,Y 343.599,Z 992.111,A -85,B 0,C 180,E1 9039.281,E2 9039.281} C_VEL
LIN {X 0,Y 349.723,Z 971.346,A -85,B 0,C 180,E1 9037.766,E2 9037.766} C_VEL
LIN {X 0,Y 354.835,Z 950.833,A -85,B 0,C 180,E1 9036.575,E2 9036.575} C_VEL
LIN {X 0,Y 359.104,Z 929.285,A -85,B 0,C 180,E1 9035.625,E2 9035.625} C_VEL
LIN {X 0,Y 362.638,Z 905.828,A -85,B 0,C 180,E1 9034.876,E2 9034.876} C_VEL
LIN {X 0,Y 363.746,Z 895.261,A -85,B 0,C 180,E1 9034.599,E2 9034.599} C_VEL
LIN {X 0,Y 361.843,Z 900.079,A -85,B 0,C 180,E1 9034.361,E2 9034.361} C_VEL
LIN {X 0,Y 357.458,Z 914.157,A -85,B 0,C 180,E1 9034.086,E2 9034.086} C_VEL
LIN {X 0,Y 352.2,Z 926.312,A -85,B 0,C 180,E1 9033.626,E2 9033.626} C_VEL
LIN {X 0,Y 346.916,Z 935.305,A -85,B 0,C 180,E1 9033.006,E2 9033.006} C_VEL
LIN {X 0,Y 343.618,Z 940.042,A -85,B 0,C 180,E1 9032.569,E2 9032.569} C_VEL
LIN {X 0,Y 337.908,Z 949.536,A -85,B 0,C 180,E1 9031.983,E2 9031.983} C_VEL
LIN {X 0,Y 332.802,Z 956.118,A -85,B 0,C 180,E1 9031.316,E2 9031.316} C_VEL
LIN {X 0,Y 328.276,Z 961.012,A -85,B 0,C 180,E1 9030.574,E2 9030.574} C_VEL
LIN {X 0,Y 323.078,Z 967.455,A -85,B 0,C 180,E1 9029.885,E2 9029.885} C_VEL
LIN {X 0,Y 317.884,Z 972.59,A -85,B 0,C 180,E1 9028.973,E2 9028.973} C_VEL
LIN {X 0,Y 315.517,Z 974.644,A -85,B 0,C 180,E1 9028.485,E2 9028.485} C_VEL
LIN {X 0,Y 310.27,Z 979.985,A -85,B 0,C 180,E1 9027.6,E2 9027.6} C_VEL
LIN {X 0,Y 305.956,Z 983.264,A -85,B 0,C 180,E1 9026.598,E2 9026.598} C_VEL
LIN {X 0,Y 304.405,Z 984.677,A -85,B 0,C 180,E1 9026.271,E2 9026.271} C_VEL
LIN {X 0,Y 300.448,Z 988.284,A -85,B 0,C 180,E1 9025.424,E2 9025.424} C_VEL
LIN {X 0,Y 297.121,Z 990.264,A -85,B 0,C 180,E1 9024.451,E2 9024.451} C_VEL
LIN {X 0,Y 292.574,Z 994.155,A -85,B 0,C 180,E1 9023.355,E2 9023.355} C_VEL
LIN {X 0,Y 289.995,Z 995.859,A -85,B 0,C 180,E1 9022.289,E2 9022.289} C_VEL
LIN {X 0,Y 289.283,Z 1000.003,A -85,B 0,C 180,E1 9021.493,E2 9021.493} C_VEL
LIN {X 0,Y 287.582,Z 1012.92,A -85,B 0,C 180,E1 9019.076,E2 9019.076} C_VEL
LIN {X 0,Y 285.978,Z 1025.128,A -85,B 0,C 180,E1 9016.243,E2 9016.243} C_VEL
LIN {X 0,Y 284.78,Z 1035.081,A -85,B 0,C 180,E1 9013.399,E2 9013.399} C_VEL
LIN {X 0,Y 283.887,Z 1043.536,A -85,B 0,C 180,E1 9010.348,E2 9010.348} C_VEL
LIN {X 0,Y 283.366,Z 1050.488,A -85,B 0,C 180,E1 9007.095,E2 9007.095} C_VEL
LIN {X 0,Y 283.227,Z 1055.549,A -85,B 0,C 180,E1 9003.847,E2 9003.847} C_VEL
LIN {X 0,Y 283.395,Z 1058.771,A -85,B 0,C 180,E1 9000.607,E2 9000.607} C_VEL
LIN {X 0,Y 283.857,Z 1060.342,A -85,B 0,C 180,E1 8997.376,E2 8997.376} C_VEL
LIN {X 0,Y 284.659,Z 1060.239,A -85,B 0,C 180,E1 8994.154,E2 8994.154} C_VEL
LIN {X 0,Y 285.853,Z 1058.375,A -85,B 0,C 180,E1 8990.945,E2 8990.945} C_VEL
LIN {X 0,Y 287.512,Z 1054.699,A -85,B 0,C 180,E1 8987.746,E2 8987.746} C_VEL
LIN {X 0,Y 289.5,Z 1049.514,A -85,B 0,C 180,E1 8984.783,E2 8984.783} C_VEL
LIN {X 0,Y 291.923,Z 1042.41,A -85,B 0,C 180,E1 8981.84,E2 8981.84} C_VEL
LIN {X 0,Y 294.793,Z 1033.052,A -85,B 0,C 180,E1 8978.93,E2 8978.93} C_VEL
LIN {X 0,Y 297.628,Z 1022.719,A -85,B 0,C 180,E1 8976.437,E2 8976.437} C_VEL
LIN {X 0,Y 300.508,Z 1010.884,A -85,B 0,C 180,E1 8974.16,E2 8974.16} C_VEL
LIN {X 0,Y 301.553,Z 1007.684,A -85,B 0,C 180,E1 8973.54,E2 8973.54} C_VEL
LIN {X 0,Y 305.199,Z 1005.645,A -85,B 0,C 180,E1 8972.7,E2 8972.7} C_VEL
LIN {X 0,Y 308.362,Z 1003.469,A -85,B 0,C 180,E1 8972.166,E2 8972.166} C_VEL
LIN {X 0,Y 312.752,Z 1000.762,A -85,B 0,C 180,E1 8971.345,E2 8971.345} C_VEL
LIN {X 0,Y 316.04,Z 998.238,A -85,B 0,C 180,E1 8970.843,E2 8970.843} C_VEL
LIN {X 0,Y 320.727,Z 995.058,A -85,B 0,C 180,E1 8970.08,E2 8970.08} C_VEL
LIN {X 0,Y 325.142,Z 991.432,A -85,B 0,C 180,E1 8969.51,E2 8969.51} C_VEL
LIN {X 0,Y 331.023,Z 986.735,A -85,B 0,C 180,E1 8968.7,E2 8968.7} C_VEL
LIN {X 0,Y 335.694,Z 982.267,A -85,B 0,C 180,E1 8968.185,E2 8968.185} C_VEL
LIN {X 0,Y 342.023,Z 976.523,A -85,B 0,C 180,E1 8967.46,E2 8967.46} C_VEL
LIN {X 0,Y 347.965,Z 969.81,A -85,B 0,C 180,E1 8966.911,E2 8966.911} C_VEL
LIN {X 0,Y 351.141,Z 966.614,A -85,B 0,C 180,E1 8966.579,E2 8966.579} C_VEL
LIN {X 0,Y 345.407,Z 987.401,A -85,B 0,C 180,E1 8965.151,E2 8965.151} C_VEL
LIN {X 0,Y 338.821,Z 1008.223,A -85,B 0,C 180,E1 8963.386,E2 8963.386} C_VEL
LIN {X 0,Y 332.041,Z 1027.639,A -85,B 0,C 180,E1 8961.391,E2 8961.391} C_VEL
LIN {X 0,Y 325.139,Z 1045.493,A -85,B 0,C 180,E1 8959.156,E2 8959.156} C_VEL
LIN {X 0,Y 318.05,Z 1062.906,A -85,B 0,C 180,E1 8956.569,E2 8956.569} C_VEL
LIN {X 0,Y 311.084,Z 1079.042,A -85,B 0,C 180,E1 8953.684,E2 8953.684} C_VEL
LIN {X 0,Y 303.866,Z 1095.43,A -85,B 0,C 180,E1 8950.161,E2 8950.161} C_VEL
LIN {X 0,Y 297.638,Z 1109.662,A -85,B 0,C 180,E1 8946.484,E2 8946.484} C_VEL
LIN {X 0,Y 292.196,Z 1122.32,A -85,B 0,C 180,E1 8942.496,E2 8942.496} C_VEL
LIN {X 0,Y 287.515,Z 1134.098,A -85,B 0,C 180,E1 8938,E2 8938} C_VEL
LIN {X 0,Y 284.253,Z 1143.462,A -85,B 0,C 180,E1 8933.641,E2 8933.641} C_VEL
LIN {X 0,Y 282.033,Z 1150.938,A -85,B 0,C 180,E1 8929.251,E2 8929.251} C_VEL
LIN {X 0,Y 280.732,Z 1156.933,A -85,B 0,C 180,E1 8924.859,E2 8924.859} C_VEL
LIN {X 0,Y 280.123,Z 1161.216,A -85,B 0,C 180,E1 8920.489,E2 8920.489} C_VEL
LIN {X 0,Y 279.974,Z 1163.769,A -85,B 0,C 180,E1 8916.768,E2 8916.768} C_VEL
LIN {X 0,Y 279.969,Z 1165.37,A -85,B 0,C 180,E1 8912.456,E2 8912.456} C_VEL
LIN {X 0,Y 279.975,Z 1165.516,A -85,B 0,C 180,E1 8908.772,E2 8908.772} C_VEL
LIN {X 0,Y 279.963,Z 1164.616,A -85,B 0,C 180,E1 8905.083,E2 8905.083} C_VEL
LIN {X 0,Y 280.064,Z 1162.227,A -85,B 0,C 180,E1 8900.755,E2 8900.755} C_VEL
LIN {X 0,Y 280.465,Z 1158.47,A -85,B 0,C 180,E1 8896.601,E2 8896.601} C_VEL
LIN {X 0,Y 281.55,Z 1153.019,A -85,B 0,C 180,E1 8892.125,E2 8892.125} C_VEL
LIN {X 0,Y 283.388,Z 1146.073,A -85,B 0,C 180,E1 8887.82,E2 8887.82} C_VEL
LIN {X 0,Y 286.356,Z 1137.234,A -85,B 0,C 180,E1 8883.361,E2 8883.361} C_VEL
LIN {X 0,Y 290.112,Z 1127.378,A -85,B 0,C 180,E1 8879.331,E2 8879.331} C_VEL
LIN {X 0,Y 295.51,Z 1114.452,A -85,B 0,C 180,E1 8874.965,E2 8874.965} C_VEL
LIN {X 0,Y 301.451,Z 1100.934,A -85,B 0,C 180,E1 8871.18,E2 8871.18} C_VEL
LIN {X 0,Y 307.997,Z 1086.005,A -85,B 0,C 180,E1 8867.744,E2 8867.744} C_VEL
LIN {X 0,Y 315.545,Z 1068.6,A -85,B 0,C 180,E1 8864.408,E2 8864.408} C_VEL
LIN {X 0,Y 322.861,Z 1051.185,A -85,B 0,C 180,E1 8861.641,E2 8861.641} C_VEL
LIN {X 0,Y 329.909,Z 1033.055,A -85,B 0,C 180,E1 8859.268,E2 8859.268} C_VEL
LIN {X 0,Y 336.882,Z 1013.849,A -85,B 0,C 180,E1 8857.164,E2 8857.164} C_VEL
LIN {X 0,Y 343.113,Z 994.739,A -85,B 0,C 180,E1 8855.443,E2 8855.443} C_VEL
LIN {X 0,Y 349.55,Z 972.387,A -85,B 0,C 180,E1 8853.803,E2 8853.803} C_VEL
LIN {X 0,Y 354.781,Z 951.331,A -85,B 0,C 180,E1 8852.566,E2 8852.566} C_VEL
LIN {X 0,Y 359.283,Z 928.846,A -85,B 0,C 180,E1 8851.546,E2 8851.546} C_VEL
LIN {X 0,Y 362.974,Z 905.474,A -85,B 0,C 180,E1 8850.756,E2 8850.756} C_VEL
LIN {X 0,Y 365.345,Z 882.873,A -85,B 0,C 180,E1 8850.198,E2 8850.198} C_VEL
LIN {X 0,Y 379.827,Z 676.646,A -85,B 0,C 180,E1 8845.981,E2 8845.981} C_VEL
LIN {X 0,Y 380.255,Z 669.056,A -85,B 0,C 180,E1 8845.796,E2 8845.796} C_VEL
LIN {X 0,Y 372.615,Z 656.653,A -85,B 0,C 180,E1 8842.981,E2 8842.981} C_VEL
LIN {X 0,Y 365.67,Z 646.165,A -85,B 0,C 180,E1 8840.069,E2 8840.069} C_VEL
LIN {X 0,Y 360.082,Z 638.193,A -85,B 0,C 180,E1 8837.367,E2 8837.367} C_VEL
LIN {X 0,Y 356.051,Z 632.762,A -85,B 0,C 180,E1 8835.139,E2 8835.139} C_VEL
LIN {X 0,Y 353.542,Z 629.423,A -85,B 0,C 180,E1 8833.575,E2 8833.575} C_VEL
LIN {X 0,Y 350.091,Z 624.913,A -85,B 0,C 180,E1 8831.115,E2 8831.115} C_VEL
LIN {X 0,Y 345.921,Z 619.674,A -85,B 0,C 180,E1 8827.306,E2 8827.306} C_VEL
LIN {X 0,Y 341.863,Z 615.312,A -85,B 0,C 180,E1 8820.67,E2 8820.67} C_VEL
LIN {X 0,Y 341.356,Z 614.91,A -85,B 0,C 180,E1 8817.481,E2 8817.481} C_VEL
LIN {X 0,Y 341.888,Z 616.635,A -85,B 0,C 180,E1 8813.619,E2 8813.619} C_VEL
LIN {X 0,Y 344.153,Z 619.638,A -85,B 0,C 180,E1 8809.368,E2 8809.368} C_VEL
LIN {X 0,Y 347.701,Z 624.921,A -85,B 0,C 180,E1 8805.426,E2 8805.426} C_VEL
LIN {X 0,Y 351.362,Z 630.534,A -85,B 0,C 180,E1 8802.443,E2 8802.443} C_VEL
LIN {X 0,Y 354.426,Z 635.077,A -85,B 0,C 180,E1 8800.384,E2 8800.384} C_VEL
LIN {X 0,Y 359.08,Z 642.073,A -85,B 0,C 180,E1 8797.704,E2 8797.704} C_VEL
LIN {X 0,Y 365.085,Z 651.638,A -85,B 0,C 180,E1 8794.751,E2 8794.751} C_VEL
LIN {X 0,Y 372.004,Z 663.264,A -85,B 0,C 180,E1 8791.822,E2 8791.822} C_VEL
LIN {X 0,Y 377.96,Z 673.975,A -85,B 0,C 180,E1 8789.581,E2 8789.581} C_VEL
LIN {X 0,Y 363.806,Z 894.191,A -85,B 0,C 180,E1 8785.308,E2 8785.308} C_VEL
LIN {X 0,Y 361.061,Z 916.812,A -85,B 0,C 180,E1 8784.705,E2 8784.705} C_VEL
LIN {X 0,Y 357.495,Z 937.851,A -85,B 0,C 180,E1 8783.929,E2 8783.929} C_VEL
LIN {X 0,Y 353.204,Z 957.37,A -85,B 0,C 180,E1 8782.968,E2 8782.968} C_VEL
LIN {X 0,Y 347.84,Z 977.872,A -85,B 0,C 180,E1 8781.696,E2 8781.696} C_VEL
LIN {X 0,Y 342.077,Z 996.653,A -85,B 0,C 180,E1 8780.24,E2 8780.24} C_VEL
LIN {X 0,Y 335.443,Z 1015.598,A -85,B 0,C 180,E1 8778.431,E2 8778.431} C_VEL
LIN {X 0,Y 328.661,Z 1033.21,A -85,B 0,C 180,E1 8776.39,E2 8776.39} C_VEL
LIN {X 0,Y 321.56,Z 1049.866,A -85,B 0,C 180,E1 8774.024,E2 8774.024} C_VEL
LIN {X 0,Y 314.142,Z 1066.192,A -85,B 0,C 180,E1 8771.212,E2 8771.212} C_VEL
LIN {X 0,Y 307.26,Z 1080.687,A -85,B 0,C 180,E1 8768.191,E2 8768.191} C_VEL
LIN {X 0,Y 300.696,Z 1093.972,A -85,B 0,C 180,E1 8764.783,E2 8764.783} C_VEL
LIN {X 0,Y 294.786,Z 1105.971,A -85,B 0,C 180,E1 8761.035,E2 8761.035} C_VEL
LIN {X 0,Y 289.897,Z 1116.314,A -85,B 0,C 180,E1 8757.082,E2 8757.082} C_VEL
LIN {X 0,Y 285.944,Z 1125.11,A -85,B 0,C 180,E1 8752.838,E2 8752.838} C_VEL
LIN {X 0,Y 283.057,Z 1132.49,A -85,B 0,C 180,E1 8748.323,E2 8748.323} C_VEL
LIN {X 0,Y 281.339,Z 1137.94,A -85,B 0,C 180,E1 8743.985,E2 8743.985} C_VEL
LIN {X 0,Y 280.446,Z 1141.733,A -85,B 0,C 180,E1 8739.646,E2 8739.646} C_VEL
LIN {X 0,Y 280.073,Z 1144.204,A -85,B 0,C 180,E1 8735.326,E2 8735.326} C_VEL
LIN {X 0,Y 280,Z 1145.16,A -85,B 0,C 180,E1 8731.228,E2 8731.228} C_VEL
LIN {X 0,Y 280.01,Z 1144.997,A -85,B 0,C 180,E1 8727.134,E2 8727.134} C_VEL
LIN {X 0,Y 280.186,Z 1143.343,A -85,B 0,C 180,E1 8722.825,E2 8722.825} C_VEL
LIN {X 0,Y 280.758,Z 1140.249,A -85,B 0,C 180,E1 8718.338,E2 8718.338} C_VEL
LIN {X 0,Y 282.016,Z 1135.646,A -85,B 0,C 180,E1 8713.946,E2 8713.946} C_VEL
LIN {X 0,Y 284.294,Z 1129.192,A -85,B 0,C 180,E1 8709.409,E2 8709.409} C_VEL
LIN {X 0,Y 287.604,Z 1121.373,A -85,B 0,C 180,E1 8705.124,E2 8705.124} C_VEL
LIN {X 0,Y 291.863,Z 1112.098,A -85,B 0,C 180,E1 8701.116,E2 8701.116} C_VEL
LIN {X 0,Y 297.262,Z 1100.989,A -85,B 0,C 180,E1 8697.212,E2 8697.212} C_VEL
LIN {X 0,Y 301.831,Z 1091.731,A -85,B 0,C 180,E1 8694.492,E2 8694.492} C_VEL
LIN {X 0,Y 303.089,Z 1087.615,A -85,B 0,C 180,E1 8693.269,E2 8693.269} C_VEL
LIN {X 0,Y 303.583,Z 1077.198,A -85,B 0,C 180,E1 8690.016,E2 8690.016} C_VEL
LIN {X 0,Y 305.183,Z 1072.595,A -85,B 0,C 180,E1 8688.879,E2 8688.879} C_VEL
LIN {X 0,Y 312.503,Z 1057.436,A -85,B 0,C 180,E1 8686.029,E2 8686.029} C_VEL
LIN {X 0,Y 320.383,Z 1040.13,A -85,B 0,C 180,E1 8683.351,E2 8683.351} C_VEL
LIN {X 0,Y 327.513,Z 1023.128,A -85,B 0,C 180,E1 8681.189,E2 8681.189} C_VEL
LIN {X 0,Y 334.506,Z 1004.532,A -85,B 0,C 180,E1 8679.27,E2 8679.27} C_VEL
LIN {X 0,Y 341.254,Z 984.315,A -85,B 0,C 180,E1 8677.575,E2 8677.575} C_VEL
LIN {X 0,Y 346.732,Z 965.289,A -85,B 0,C 180,E1 8676.294,E2 8676.294} C_VEL
LIN {X 0,Y 351.719,Z 944.449,A -85,B 0,C 180,E1 8675.185,E2 8675.185} C_VEL
LIN {X 0,Y 354.255,Z 931.435,A -85,B 0,C 180,E1 8674.605,E2 8674.605} C_VEL
LIN {X 0,Y 348.729,Z 940.3,A -85,B 0,C 180,E1 8673.994,E2 8673.994} C_VEL
LIN {X 0,Y 345.701,Z 944.559,A -85,B 0,C 180,E1 8673.633,E2 8673.633} C_VEL
LIN {X 0,Y 339.368,Z 954.458,A -85,B 0,C 180,E1 8673.029,E2 8673.029} C_VEL
LIN {X 0,Y 333.554,Z 961.711,A -85,B 0,C 180,E1 8672.293,E2 8672.293} C_VEL
LIN {X 0,Y 329.45,Z 965.863,A -85,B 0,C 180,E1 8671.672,E2 8671.672} C_VEL
LIN {X 0,Y 323.288,Z 973.138,A -85,B 0,C 180,E1 8670.891,E2 8670.891} C_VEL
LIN {X 0,Y 317.898,Z 978.223,A -85,B 0,C 180,E1 8670.006,E2 8670.006} C_VEL
LIN {X 0,Y 314.955,Z 980.735,A -85,B 0,C 180,E1 8669.477,E2 8669.477} C_VEL
LIN {X 0,Y 309.491,Z 986.001,A -85,B 0,C 180,E1 8668.564,E2 8668.564} C_VEL
LIN {X 0,Y 304.019,Z 990.085,A -85,B 0,C 180,E1 8667.379,E2 8667.379} C_VEL
LIN {X 0,Y 299.072,Z 994.282,A -85,B 0,C 180,E1 8666.401,E2 8666.401} C_VEL
LIN {X 0,Y 294.979,Z 996.822,A -85,B 0,C 180,E1 8665.283,E2 8665.283} C_VEL
LIN {X 0,Y 290.637,Z 1000.392,A -85,B 0,C 180,E1 8664.263,E2 8664.263} C_VEL
LIN {X 0,Y 286.828,Z 1002.49,A -85,B 0,C 180,E1 8663.032,E2 8663.032} C_VEL
LIN {X 0,Y 283.059,Z 1005.33,A -85,B 0,C 180,E1 8661.989,E2 8661.989} C_VEL
LIN {X 0,Y 280.931,Z 1006.513,A -85,B 0,C 180,E1 8660.959,E2 8660.959} C_VEL
LIN {X 0,Y 278.551,Z 1023.08,A -85,B 0,C 180,E1 8657.29,E2 8657.29} C_VEL
LIN {X 0,Y 277.218,Z 1033.578,A -85,B 0,C 180,E1 8654.411,E2 8654.411} C_VEL
LIN {X 0,Y 276.149,Z 1043.113,A -85,B 0,C 180,E1 8651.121,E2 8651.121} C_VEL
LIN {X 0,Y 275.542,Z 1050.451,A -85,B 0,C 180,E1 8647.845,E2 8647.845} C_VEL
LIN {X 0,Y 275.322,Z 1055.839,A -85,B 0,C 180,E1 8644.583,E2 8644.583} C_VEL
LIN {X 0,Y 275.456,Z 1059.633,A -85,B 0,C 180,E1 8641.249,E2 8641.249} C_VEL
LIN {X 0,Y 275.904,Z 1061.727,A -85,B 0,C 180,E1 8637.924,E2 8637.924} C_VEL
LIN {X 0,Y 276.69,Z 1062.064,A -85,B 0,C 180,E1 8634.609,E2 8634.609} C_VEL
LIN {X 0,Y 277.993,Z 1060.586,A -85,B 0,C 180,E1 8631.104,E2 8631.104} C_VEL
LIN {X 0,Y 279.723,Z 1057.38,A -85,B 0,C 180,E1 8627.826,E2 8627.826} C_VEL
LIN {X 0,Y 281.961,Z 1052.214,A -85,B 0,C 180,E1 8624.577,E2 8624.577} C_VEL
LIN {X 0,Y 284.537,Z 1045.489,A -85,B 0,C 180,E1 8621.564,E2 8621.564} C_VEL
LIN {X 0,Y 287.365,Z 1037.233,A -85,B 0,C 180,E1 8618.786,E2 8618.786} C_VEL
LIN {X 0,Y 290.363,Z 1027.604,A -85,B 0,C 180,E1 8616.242,E2 8616.242} C_VEL
LIN {X 0,Y 293.464,Z 1017.231,A -85,B 0,C 180,E1 8613.982,E2 8613.982} C_VEL
LIN {X 0,Y 297.213,Z 1015.392,A -85,B 0,C 180,E1 8613.062,E2 8613.062} C_VEL
LIN {X 0,Y 300.4,Z 1013.522,A -85,B 0,C 180,E1 8612.442,E2 8612.442} C_VEL
LIN {X 0,Y 304.74,Z 1011.084,A -85,B 0,C 180,E1 8611.593,E2 8611.593} C_VEL
LIN {X 0,Y 307.113,Z 1009.511,A -85,B 0,C 180,E1 8611.195,E2 8611.195} C_VEL
LIN {X 0,Y 312.525,Z 1006.222,A -85,B 0,C 180,E1 8610.272,E2 8610.272} C_VEL
LIN {X 0,Y 315.885,Z 1003.911,A -85,B 0,C 180,E1 8609.784,E2 8609.784} C_VEL
LIN {X 0,Y 321.645,Z 999.905,A -85,B 0,C 180,E1 8608.935,E2 8608.935} C_VEL
LIN {X 0,Y 326.042,Z 996.451,A -85,B 0,C 180,E1 8608.373,E2 8608.373} C_VEL
LIN {X 0,Y 332.274,Z 991.567,A -85,B 0,C 180,E1 8607.614,E2 8607.614} C_VEL
LIN {X 0,Y 336.992,Z 987.259,A -85,B 0,C 180,E1 8607.115,E2 8607.115} C_VEL
LIN {X 0,Y 341.926,Z 982.894,A -85,B 0,C 180,E1 8606.573,E2 8606.573} C_VEL
LIN {X 0,Y 335.731,Z 1002.706,A -85,B 0,C 180,E1 8604.984,E2 8604.984} C_VEL
LIN {X 0,Y 328.578,Z 1022.666,A -85,B 0,C 180,E1 8603.015,E2 8603.015} C_VEL
LIN {X 0,Y 321.044,Z 1041.949,A -85,B 0,C 180,E1 8600.708,E2 8600.708} C_VEL
LIN {X 0,Y 313.776,Z 1059.188,A -85,B 0,C 180,E1 8598.215,E2 8598.215} C_VEL
LIN {X 0,Y 306.216,Z 1076.176,A -85,B 0,C 180,E1 8595.25,E2 8595.25} C_VEL
LIN {X 0,Y 299.027,Z 1091.89,A -85,B 0,C 180,E1 8591.97,E2 8591.97} C_VEL
LIN {X 0,Y 292.544,Z 1105.714,A -85,B 0,C 180,E1 8588.466,E2 8588.466} C_VEL
LIN {X 0,Y 286.484,Z 1119.007,A -85,B 0,C 180,E1 8584.43,E2 8584.43} C_VEL
LIN {X 0,Y 281.591,Z 1130.292,A -85,B 0,C 180,E1 8580.279,E2 8580.279} C_VEL
LIN {X 0,Y 277.666,Z 1140.208,A -85,B 0,C 180,E1 8575.813,E2 8575.813} C_VEL
LIN {X 0,Y 274.941,Z 1148.375,A -85,B 0,C 180,E1 8571.325,E2 8571.325} C_VEL
LIN {X 0,Y 273.206,Z 1154.754,A -85,B 0,C 180,E1 8566.805,E2 8566.805} C_VEL
LIN {X 0,Y 272.315,Z 1159.708,A -85,B 0,C 180,E1 8562.296,E2 8562.296} C_VEL
LIN {X 0,Y 272.012,Z 1162.869,A -85,B 0,C 180,E1 8558.029,E2 8558.029} C_VEL
LIN {X 0,Y 271.97,Z 1164.619,A -85,B 0,C 180,E1 8554.217,E2 8554.217} C_VEL
LIN {X 0,Y 271.988,Z 1165.361,A -85,B 0,C 180,E1 8550,E2 8550} C_VEL
LIN {X 0,Y 271.97,Z 1164.615,A -85,B 0,C 180,E1 8545.783,E2 8545.783} C_VEL
LIN {X 0,Y 272.012,Z 1162.863,A -85,B 0,C 180,E1 8541.971,E2 8541.971} C_VEL
LIN {X 0,Y 272.341,Z 1159.48,A -85,B 0,C 180,E1 8537.49,E2 8537.49} C_VEL
LIN {X 0,Y 273.205,Z 1154.741,A -85,B 0,C 180,E1 8533.195,E2 8533.195} C_VEL
LIN {X 0,Y 274.998,Z 1148.15,A -85,B 0,C 180,E1 8528.555,E2 8528.555} C_VEL
LIN {X 0,Y 277.677,Z 1140.151,A -85,B 0,C 180,E1 8524.17,E2 8524.17} C_VEL
LIN {X 0,Y 281.804,Z 1129.728,A -85,B 0,C 180,E1 8519.511,E2 8519.511} C_VEL
LIN {X 0,Y 286.757,Z 1118.376,A -85,B 0,C 180,E1 8515.365,E2 8515.365} C_VEL
LIN {X 0,Y 292.611,Z 1105.499,A -85,B 0,C 180,E1 8511.489,E2 8511.489} C_VEL
LIN {X 0,Y 299.372,Z 1091.054,A -85,B 0,C 180,E1 8507.854,E2 8507.854} C_VEL
LIN {X 0,Y 306.423,Z 1075.622,A -85,B 0,C 180,E1 8504.656,E2 8504.656} C_VEL
LIN {X 0,Y 314.442,Z 1057.482,A -85,B 0,C 180,E1 8501.534,E2 8501.534} C_VEL
LIN {X 0,Y 322.029,Z 1039.486,A -85,B 0,C 180,E1 8498.976,E2 8498.976} C_VEL
LIN {X 0,Y 329.123,Z 1021.017,A -85,B 0,C 180,E1 8496.822,E2 8496.822} C_VEL
LIN {X 0,Y 336.298,Z 1000.694,A -85,B 0,C 180,E1 8494.856,E2 8494.856} C_VEL
LIN {X 0,Y 342.294,Z 981.484,A -85,B 0,C 180,E1 8493.34,E2 8493.34} C_VEL
LIN {X 0,Y 348.2,Z 959.725,A -85,B 0,C 180,E1 8491.948,E2 8491.948} C_VEL
LIN {X 0,Y 352.841,Z 939.477,A -85,B 0,C 180,E1 8490.916,E2 8490.916} C_VEL
LIN {X 0,Y 356.947,Z 917.078,A -85,B 0,C 180,E1 8490.044,E2 8490.044} C_VEL
LIN {X 0,Y 360.092,Z 894.249,A -85,B 0,C 180,E1 8489.383,E2 8489.383} C_VEL
LIN {X 0,Y 365.432,Z 822.472,A -85,B 0,C 180,E1 8487.874,E2 8487.874} C_VEL
LIN {X 0,Y 376.222,Z 673.658,A -85,B 0,C 180,E1 8484.828,E2 8484.828} C_VEL
LIN {X 0,Y 369.662,Z 662.832,A -85,B 0,C 180,E1 8482.293,E2 8482.293} C_VEL
LIN {X 0,Y 363.338,Z 653.035,A -85,B 0,C 180,E1 8479.533,E2 8479.533} C_VEL
LIN {X 0,Y 358.048,Z 645.34,A -85,B 0,C 180,E1 8476.883,E2 8476.883} C_VEL
LIN {X 0,Y 352.917,Z 638.055,A -85,B 0,C 180,E1 8473.851,E2 8473.851} C_VEL
LIN {X 0,Y 348.579,Z 632.499,A -85,B 0,C 180,E1 8470.745,E2 8470.745} C_VEL
LIN {X 0,Y 344.778,Z 627.544,A -85,B 0,C 180,E1 8467.163,E2 8467.163} C_VEL
LIN {X 0,Y 340.886,Z 623.27,A -85,B 0,C 180,E1 8460.672,E2 8460.672} C_VEL
LIN {X 0,Y 340.388,Z 622.83,A -85,B 0,C 180,E1 8457.643,E2 8457.643} C_VEL
LIN {X 0,Y 340.863,Z 624.52,A -85,B 0,C 180,E1 8453.769,E2 8453.769} C_VEL
LIN {X 0,Y 343.013,Z 627.465,A -85,B 0,C 180,E1 8449.588,E2 8449.588} C_VEL
LIN {X 0,Y 346.467,Z 632.806,A -85,B 0,C 180,E1 8445.629,E2 8445.629} C_VEL
LIN {X 0,Y 349.853,Z 638.095,A -85,B 0,C 180,E1 8442.794,E2 8442.794} C_VEL
LIN {X 0,Y 352.837,Z 642.661,A -85,B 0,C 180,E1 8440.723,E2 8440.723} C_VEL
LIN {X 0,Y 357.398,Z 649.66,A -85,B 0,C 180,E1 8438.026,E2 8438.026} C_VEL
LIN {X 0,Y 363.45,Z 659.636,A -85,B 0,C 180,E1 8434.977,E2 8434.977} C_VEL
LIN {X 0,Y 369.761,Z 670.534,A -85,B 0,C 180,E1 8432.239,E2 8432.239} C_VEL
LIN {X 0,Y 373.973,Z 678.314,A -85,B 0,C 180,E1 8430.584,E2 8430.584} C_VEL
LIN {X 0,Y 359.485,Z 895.166,A -85,B 0,C 180,E1 8426.366,E2 8426.366} C_VEL
LIN {X 0,Y 356.641,Z 917.443,A -85,B 0,C 180,E1 8425.765,E2 8425.765} C_VEL
LIN {X 0,Y 352.872,Z 938.745,A -85,B 0,C 180,E1 8424.973,E2 8424.973} C_VEL
LIN {X 0,Y 348.464,Z 958.143,A -85,B 0,C 180,E1 8424.013,E2 8424.013} C_VEL
LIN {X 0,Y 342.637,Z 979.477,A -85,B 0,C 180,E1 8422.673,E2 8422.673} C_VEL
LIN {X 0,Y 336.429,Z 998.986,A -85,B 0,C 180,E1 8421.138,E2 8421.138} C_VEL
LIN {X 0,Y 329.599,Z 1017.52,A -85,B 0,C 180,E1 8419.323,E2 8419.323} C_VEL
LIN {X 0,Y 322.086,Z 1036.015,A -85,B 0,C 180,E1 8417.107,E2 8417.107} C_VEL
LIN {X 0,Y 314.576,Z 1052.981,A -85,B 0,C 180,E1 8414.623,E2 8414.623} C_VEL
LIN {X 0,Y 307.176,Z 1068.366,A -85,B 0,C 180,E1 8411.857,E2 8411.857} C_VEL
LIN {X 0,Y 299.691,Z 1083.285,A -85,B 0,C 180,E1 8408.601,E2 8408.601} C_VEL
LIN {X 0,Y 293.143,Z 1096.049,A -85,B 0,C 180,E1 8405.2,E2 8405.2} C_VEL
LIN {X 0,Y 287.214,Z 1107.421,A -85,B 0,C 180,E1 8401.471,E2 8401.471} C_VEL
LIN {X 0,Y 281.941,Z 1117.952,A -85,B 0,C 180,E1 8397.225,E2 8397.225} C_VEL
LIN {X 0,Y 277.927,Z 1126.584,A -85,B 0,C 180,E1 8392.864,E2 8392.864} C_VEL
LIN {X 0,Y 275.106,Z 1133.37,A -85,B 0,C 180,E1 8388.433,E2 8388.433} C_VEL
LIN {X 0,Y 273.28,Z 1138.841,A -85,B 0,C 180,E1 8383.758,E2 8383.758} C_VEL
LIN {X 0,Y 272.437,Z 1142.329,A -85,B 0,C 180,E1 8379.506,E2 8379.506} C_VEL
LIN {X 0,Y 272.069,Z 1144.622,A -85,B 0,C 180,E1 8375.06,E2 8375.06} C_VEL
LIN {X 0,Y 272.005,Z 1145.477,A -85,B 0,C 180,E1 8371.006,E2 8371.006} C_VEL
LIN {X 0,Y 272.024,Z 1145.164,A -85,B 0,C 180,E1 8366.628,E2 8366.628} C_VEL
LIN {X 0,Y 272.216,Z 1143.53,A -85,B 0,C 180,E1 8362.402,E2 8362.402} C_VEL
LIN {X 0,Y 272.899,Z 1140.303,A -85,B 0,C 180,E1 8357.731,E2 8357.731} C_VEL
LIN {X 0,Y 274.287,Z 1135.704,A -85,B 0,C 180,E1 8353.263,E2 8353.263} C_VEL
LIN {X 0,Y 276.799,Z 1129.159,A -85,B 0,C 180,E1 8348.602,E2 8348.602} C_VEL
LIN {X 0,Y 280.391,Z 1121.245,A -85,B 0,C 180,E1 8344.212,E2 8344.212} C_VEL
LIN {X 0,Y 285.073,Z 1111.715,A -85,B 0,C 180,E1 8340.035,E2 8340.035} C_VEL
LIN {X 0,Y 290.721,Z 1100.7,A -85,B 0,C 180,E1 8336.14,E2 8336.14} C_VEL
LIN {X 0,Y 297.283,Z 1088.122,A -85,B 0,C 180,E1 8332.5,E2 8332.5} C_VEL
LIN {X 0,Y 304.019,Z 1074.845,A -85,B 0,C 180,E1 8329.369,E2 8329.369} C_VEL
LIN {X 0,Y 305.183,Z 1072.595,A -85,B 0,C 180,E1 8328.879,E2 8328.879} C_VEL
LIN {X 0,Y 306.868,Z 1067.877,A -85,B 0,C 180,E1 8327.767,E2 8327.767} C_VEL
LIN {X 0,Y 308.402,Z 1055.901,A -85,B 0,C 180,E1 8324.767,E2 8324.767} C_VEL
LIN {X 0,Y 310.204,Z 1050.584,A -85,B 0,C 180,E1 8323.776,E2 8323.776} C_VEL
LIN {X 0,Y 317.837,Z 1033.974,A -85,B 0,C 180,E1 8321.385,E2 8321.385} C_VEL
LIN {X 0,Y 325.269,Z 1016.055,A -85,B 0,C 180,E1 8319.29,E2 8319.29} C_VEL
LIN {X 0,Y 332.475,Z 996.753,A -85,B 0,C 180,E1 8317.445,E2 8317.445} C_VEL
LIN {X 0,Y 338.689,Z 977.719,A -85,B 0,C 180,E1 8315.979,E2 8315.979} C_VEL
LIN {X 0,Y 344.476,Z 956.75,A -85,B 0,C 180,E1 8314.692,E2 8314.692} C_VEL
LIN {X 0,Y 345.37,Z 953.035,A -85,B 0,C 180,E1 8314.481,E2 8314.481} C_VEL
LIN {X 0,Y 338.652,Z 962.31,A -85,B 0,C 180,E1 8313.817,E2 8313.817} C_VEL
LIN {X 0,Y 332.218,Z 969.262,A -85,B 0,C 180,E1 8313.008,E2 8313.008} C_VEL
LIN {X 0,Y 329.258,Z 972.42,A -85,B 0,C 180,E1 8312.617,E2 8312.617} C_VEL
LIN {X 0,Y 322.637,Z 979.553,A -85,B 0,C 180,E1 8311.792,E2 8311.792} C_VEL
LIN {X 0,Y 316.434,Z 984.958,A -85,B 0,C 180,E1 8310.79,E2 8310.79} C_VEL
